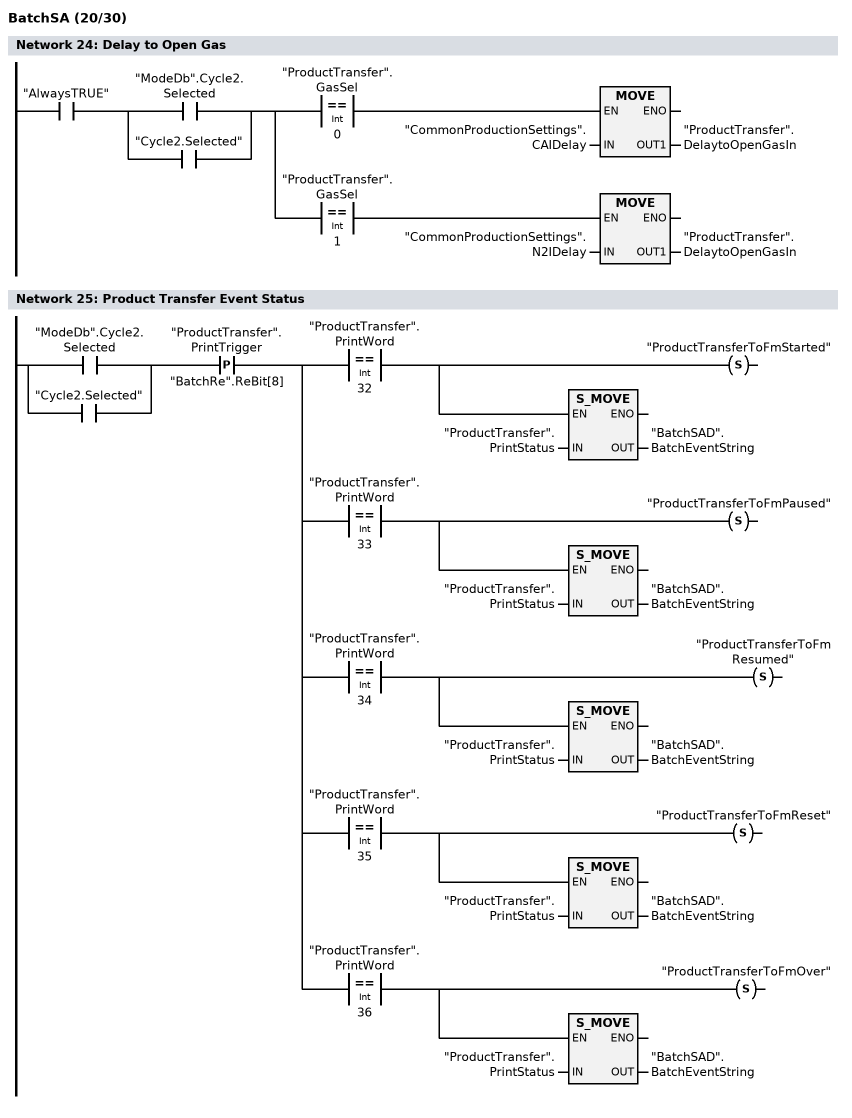
   RUNG wire#powerrail
      Contact( "AlwaysTRUE" )
      wire#w1
      Contact( "ModeDb".Cycle2.Selected )
      wire#w2
      { S7_Templates := "SrcType := Int" } EQ_Contact(in1 := "ProductTransfer".GasSel, in2 := 0)
      Move(in := "CommonProductionSettings".CAIDelay, out1 => "ProductTransfer".DelaytoOpenGasIn)
   END_RUNG
   RUNG wire#w1
      Contact( "Cycle2.Selected" )
   END_RUNG wire#w2
   RUNG wire#w2
      { S7_Templates := "SrcType := Int" } EQ_Contact(in1 := "ProductTransfer".GasSel, in2 := 1)
      Move(in := "CommonProductionSettings".N2IDelay, out1 => "ProductTransfer".DelaytoOpenGasIn)
   END_RUNG
   // the same network as SCL:
   #_w1 := "AlwaysTRUE" AND ("ModeDb".Cycle2.Selected OR "Cycle2.Selected");
   IF #_w1 AND ("ProductTransfer".GasSel = 0) THEN
       "ProductTransfer".DelaytoOpenGasIn := "CommonProductionSettings".CAIDelay;
   END_IF;
   IF #_w1 AND ("ProductTransfer".GasSel = 1) THEN
       "ProductTransfer".DelaytoOpenGasIn := "CommonProductionSettings".N2IDelay;
   END_IF;
END_REGION

REGION Network 25: Product Transfer Event Status
   RUNG wire#powerrail
      Contact( "ModeDb".Cycle2.Selected )
      wire#w1
      P_Contact(operand := "ProductTransfer".PrintTrigger, bit := "BatchRe".ReBit[8])
      wire#w2
      { S7_Templates := "SrcType := Int" } EQ_Contact(in1 := "ProductTransfer".PrintWord, in2 := 32)
      wire#w3
      S_Coil( "ProductTransferToFmStarted" )
   END_RUNG
   RUNG wire#powerrail
      Contact( "Cycle2.Selected" )
   END_RUNG wire#w1
   RUNG wire#w3
      S_Move(in := "ProductTransfer".PrintStatus, out => "BatchSAD".BatchEventString)
   END_RUNG
   RUNG wire#w2
      { S7_Templates := "SrcType := Int" } EQ_Contact(in1 := "ProductTransfer".PrintWord, in2 := 33)
      wire#w4
      S_Coil( "ProductTransferToFmPaused" )
   END_RUNG
   RUNG wire#w4
      S_Move(in := "ProductTransfer".PrintStatus, out => "BatchSAD".BatchEventString)
   END_RUNG
   RUNG wire#w2
      { S7_Templates := "SrcType := Int" } EQ_Contact(in1 := "ProductTransfer".PrintWord, in2 := 34)
      wire#w5
      S_Coil( "ProductTransferToFmResumed" )
   END_RUNG
   RUNG wire#w5
      S_Move(in := "ProductTransfer".PrintStatus, out => "BatchSAD".BatchEventString)
   END_RUNG
   RUNG wire#w2
      { S7_Templates := "SrcType := Int" } EQ_Contact(in1 := "ProductTransfer".PrintWord, in2 := 35)
      wire#w6
      S_Coil( "ProductTransferToFmReset" )
   END_RUNG
   RUNG wire#w6
      S_Move(in := "ProductTransfer".PrintStatus, out => "BatchSAD".BatchEventString)
   END_RUNG
   RUNG wire#w2
      { S7_Templates := "SrcType := Int" } EQ_Contact(in1 := "ProductTransfer".PrintWord, in2 := 36)
      wire#w7
      S_Coil( "ProductTransferToFmOver" )
   END_RUNG
   RUNG wire#w7
      S_Move(in := "ProductTransfer".PrintStatus, out => "BatchSAD".BatchEventString)
   END_RUNG
   // the same network as SCL:
   #_w1 := ("ModeDb".Cycle2.Selected OR "Cycle2.Selected") AND "ProductTransfer".PrintTrigger AND NOT "BatchRe".ReBit[8];   // rising edge of "ProductTransfer".PrintTrigger
   "BatchRe".ReBit[8] := "ProductTransfer".PrintTrigger;
   IF #_w1 AND ("ProductTransfer".PrintWord = 32) THEN
       "ProductTransferToFmStarted" := TRUE;
       "BatchSAD".BatchEventString := "ProductTransfer".PrintStatus;
   END_IF;
   IF #_w1 AND ("ProductTransfer".PrintWord = 33) THEN
       "ProductTransferToFmPaused" := TRUE;
       "BatchSAD".BatchEventString := "ProductTransfer".PrintStatus;
   END_IF;
   IF #_w1 AND ("ProductTransfer".PrintWord = 34) THEN
       "ProductTransferToFmResumed" := TRUE;
       "BatchSAD".BatchEventString := "ProductTransfer".PrintStatus;
   END_IF;
   IF #_w1 AND ("ProductTransfer".PrintWord = 35) THEN
       "ProductTransferToFmReset" := TRUE;
       "BatchSAD".BatchEventString := "ProductTransfer".PrintStatus;
   END_IF;
   IF #_w1 AND ("ProductTransfer".PrintWord = 36) THEN
       "ProductTransferToFmOver" := TRUE;
       "BatchSAD".BatchEventString := "ProductTransfer".PrintStatus;
   END_IF;
END_REGION

REGION Network 26: ******************************Jacket Vent******************************
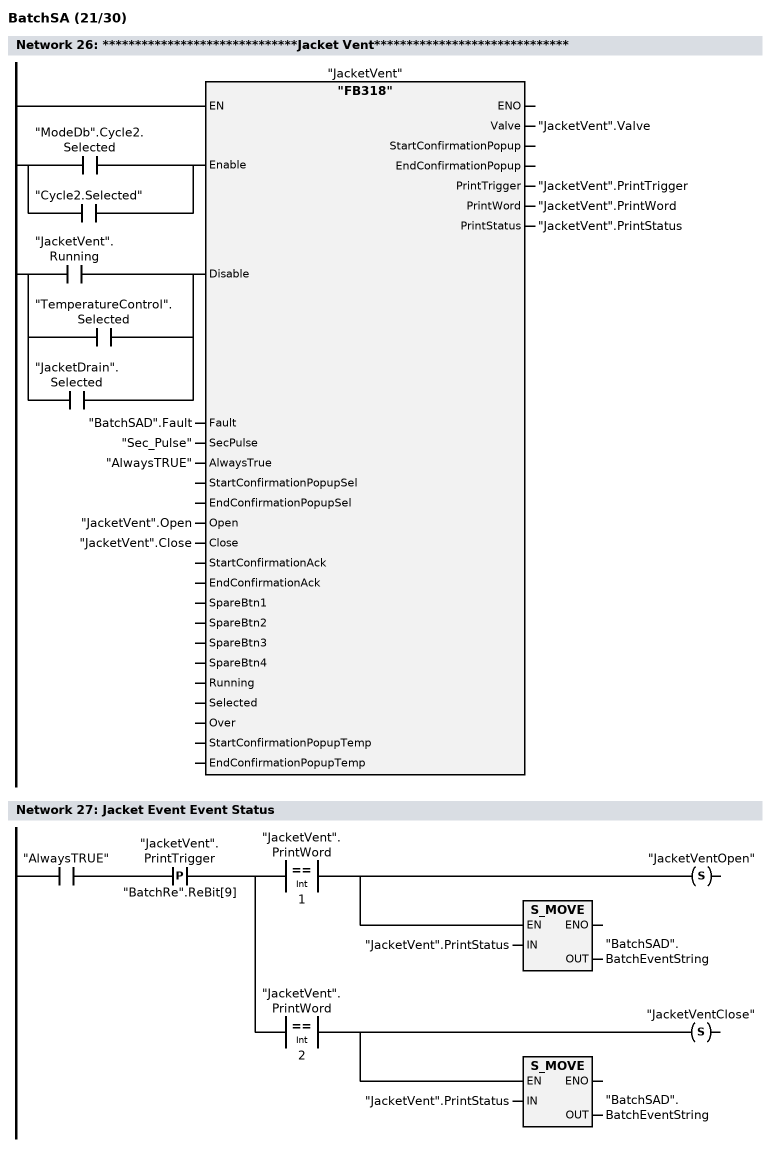
   RUNG wire#powerrail
      "JacketVent"(Enable := wire#w1, Disable := wire#w2, Fault := "BatchSAD".Fault, SecPulse := "Sec_Pulse", AlwaysTrue := "AlwaysTRUE", StartConfirmationPopupSel :=, EndConfirmationPopupSel :=, Open := "JacketVent".Open, Close := "JacketVent".Close, StartConfirmationAck :=, EndConfirmationAck :=, SpareBtn1 :=, SpareBtn2 :=, SpareBtn3 :=, SpareBtn4 :=, Running :=, Selected :=, Over :=, StartConfirmationPopupTemp :=, EndConfirmationPopupTemp :=, Valve => "JacketVent".Valve, StartConfirmationPopup =>, EndConfirmationPopup =>, PrintTrigger => "JacketVent".PrintTrigger, PrintWord => "JacketVent".PrintWord, PrintStatus => "JacketVent".PrintStatus)
   END_RUNG
   RUNG wire#powerrail
      Contact( "ModeDb".Cycle2.Selected )
   END_RUNG wire#w1
   RUNG wire#powerrail
      Contact( "Cycle2.Selected" )
   END_RUNG wire#w1
   RUNG wire#powerrail
      Contact( "JacketVent".Running )
   END_RUNG wire#w2
   RUNG wire#powerrail
      Contact( "TemperatureControl".Selected )
   END_RUNG wire#w2
   RUNG wire#powerrail
      Contact( "JacketDrain".Selected )
   END_RUNG wire#w2
   // the same network as SCL:
   "JacketVent"(Enable := "ModeDb".Cycle2.Selected OR "Cycle2.Selected",   // "FB318"
                Disable := "JacketVent".Running OR "TemperatureControl".Selected OR "JacketDrain".Selected,
                Fault := "BatchSAD".Fault,
                SecPulse := "Sec_Pulse",
                AlwaysTrue := "AlwaysTRUE",
                Open := "JacketVent".Open,
                Close := "JacketVent".Close,
                Valve => "JacketVent".Valve,
                PrintTrigger => "JacketVent".PrintTrigger,
                PrintWord => "JacketVent".PrintWord,
                PrintStatus => "JacketVent".PrintStatus);
END_REGION

REGION Network 27: Jacket Event Event Status
   RUNG wire#powerrail
      Contact( "AlwaysTRUE" )
      P_Contact(operand := "JacketVent".PrintTrigger, bit := "BatchRe".ReBit[9])
      wire#w1
      { S7_Templates := "SrcType := Int" } EQ_Contact(in1 := "JacketVent".PrintWord, in2 := 1)
      wire#w2
      S_Coil( "JacketVentOpen" )
   END_RUNG
   RUNG wire#w2
      S_Move(in := "JacketVent".PrintStatus, out => "BatchSAD".BatchEventString)
   END_RUNG
   RUNG wire#w1
      { S7_Templates := "SrcType := Int" } EQ_Contact(in1 := "JacketVent".PrintWord, in2 := 2)
      wire#w3
      S_Coil( "JacketVentClose" )
   END_RUNG
   RUNG wire#w3
      S_Move(in := "JacketVent".PrintStatus, out => "BatchSAD".BatchEventString)
   END_RUNG
   // the same network as SCL:
   #_w1 := "AlwaysTRUE" AND "JacketVent".PrintTrigger AND NOT "BatchRe".ReBit[9];   // rising edge of "JacketVent".PrintTrigger
   "BatchRe".ReBit[9] := "JacketVent".PrintTrigger;
   IF #_w1 AND ("JacketVent".PrintWord = 1) THEN
       "JacketVentOpen" := TRUE;
       "BatchSAD".BatchEventString := "JacketVent".PrintStatus;
   END_IF;
   IF #_w1 AND ("JacketVent".PrintWord = 2) THEN
       "JacketVentClose" := TRUE;
       "BatchSAD".BatchEventString := "JacketVent".PrintStatus;
   END_IF;
END_REGION

REGION Network 28: ******************************Jacket Drain******************************
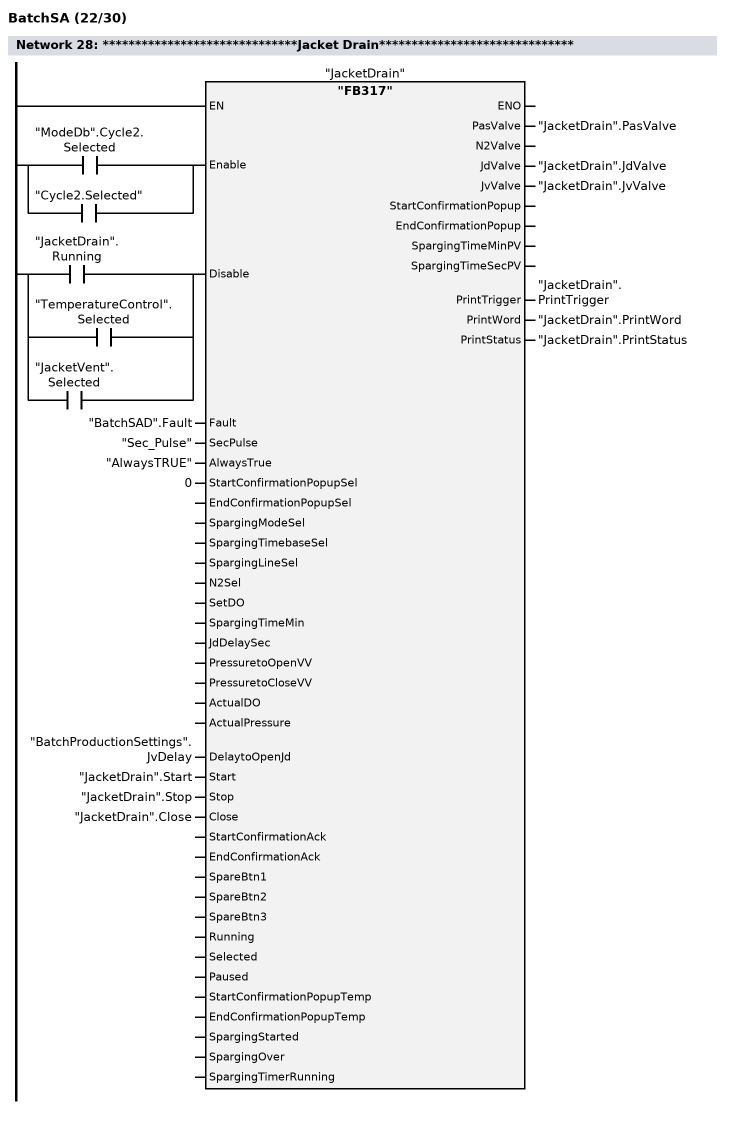
   RUNG wire#powerrail
      "JacketDrain"(Enable := wire#w1, Disable := wire#w2, Fault := "BatchSAD".Fault, SecPulse := "Sec_Pulse", AlwaysTrue := "AlwaysTRUE", StartConfirmationPopupSel := 0, EndConfirmationPopupSel :=, SpargingModeSel :=, SpargingTimebaseSel :=, SpargingLineSel :=, N2Sel :=, SetDO :=, SpargingTimeMin :=, JdDelaySec :=, PressuretoOpenVV :=, PressuretoCloseVV :=, ActualDO :=, ActualPressure :=, DelaytoOpenJd := "BatchProductionSettings".JvDelay, Start := "JacketDrain".Start, Stop := "JacketDrain".Stop, Close := "JacketDrain".Close, StartConfirmationAck :=, EndConfirmationAck :=, SpareBtn1 :=, SpareBtn2 :=, SpareBtn3 :=, Running :=, Selected :=, Paused :=, StartConfirmationPopupTemp :=, EndConfirmationPopupTemp :=, SpargingStarted :=, SpargingOver :=, SpargingTimerRunning :=, PasValve => "JacketDrain".PasValve, N2Valve =>, JdValve => "JacketDrain".JdValve, JvValve => "JacketDrain".JvValve, StartConfirmationPopup =>, EndConfirmationPopup =>, SpargingTimeMinPV =>, SpargingTimeSecPV =>, PrintTrigger => "JacketDrain".PrintTrigger, PrintWord => "JacketDrain".PrintWord, PrintStatus => "JacketDrain".PrintStatus)
   END_RUNG
   RUNG wire#powerrail
      Contact( "ModeDb".Cycle2.Selected )
   END_RUNG wire#w1
   RUNG wire#powerrail
      Contact( "Cycle2.Selected" )
   END_RUNG wire#w1
   RUNG wire#powerrail
      Contact( "JacketDrain".Running )
   END_RUNG wire#w2
   RUNG wire#powerrail
      Contact( "TemperatureControl".Selected )
   END_RUNG wire#w2
   RUNG wire#powerrail
      Contact( "JacketVent".Selected )
   END_RUNG wire#w2
   // the same network as SCL:
   "JacketDrain"(Enable := "ModeDb".Cycle2.Selected OR "Cycle2.Selected",   // "FB317"
                 Disable := "JacketDrain".Running OR "TemperatureControl".Selected OR "JacketVent".Selected,
                 Fault := "BatchSAD".Fault,
                 SecPulse := "Sec_Pulse",
                 AlwaysTrue := "AlwaysTRUE",
                 StartConfirmationPopupSel := 0,
                 DelaytoOpenJd := "BatchProductionSettings".JvDelay,
                 Start := "JacketDrain".Start,
                 Stop := "JacketDrain".Stop,
                 Close := "JacketDrain".Close,
                 PasValve => "JacketDrain".PasValve,
                 JdValve => "JacketDrain".JdValve,
                 JvValve => "JacketDrain".JvValve,
                 PrintTrigger => "JacketDrain".PrintTrigger,
                 PrintWord => "JacketDrain".PrintWord,
                 PrintStatus => "JacketDrain".PrintStatus);
END_REGION

REGION Network 29: Jacket Drain Event Status
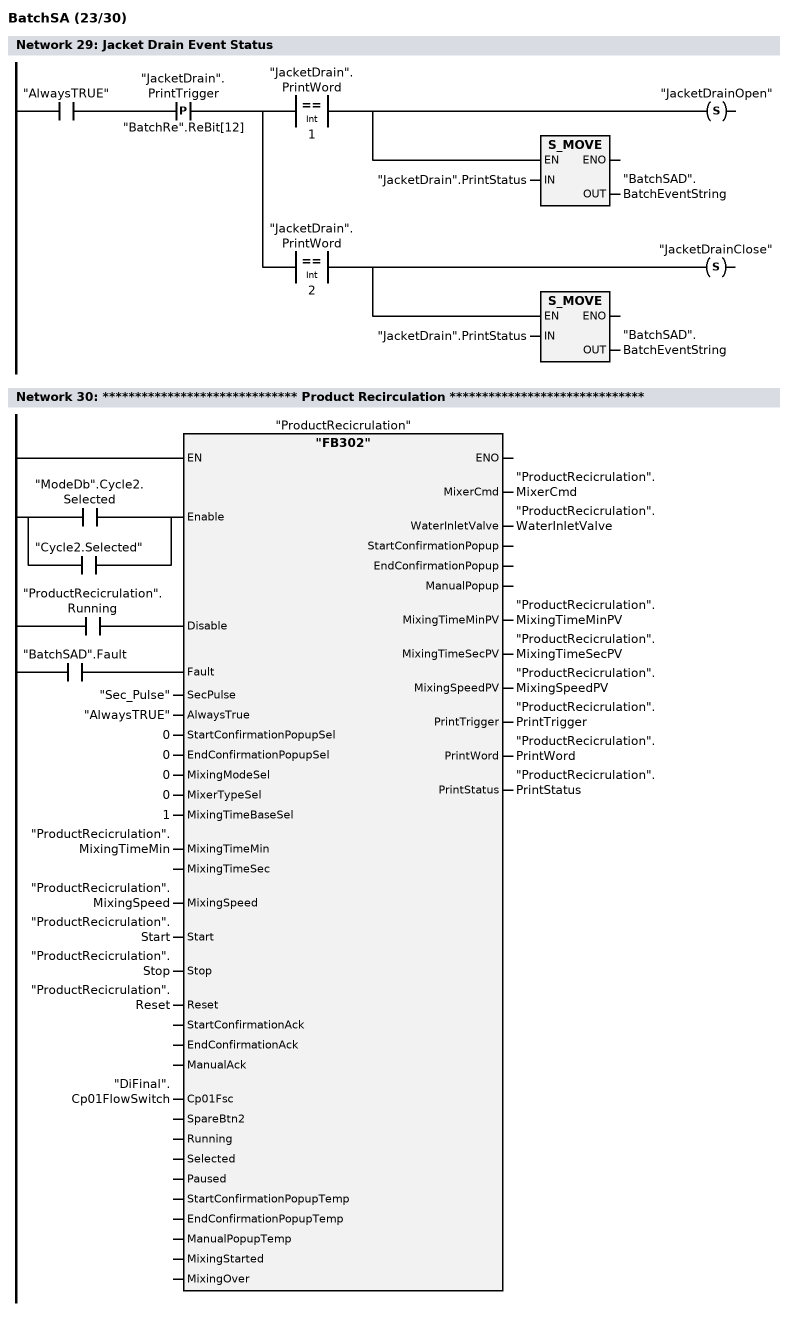
   RUNG wire#powerrail
      Contact( "AlwaysTRUE" )
      P_Contact(operand := "JacketDrain".PrintTrigger, bit := "BatchRe".ReBit[12])
      wire#w1
      { S7_Templates := "SrcType := Int" } EQ_Contact(in1 := "JacketDrain".PrintWord, in2 := 1)
      wire#w2
      S_Coil( "JacketDrainOpen" )
   END_RUNG
   RUNG wire#w2
      S_Move(in := "JacketDrain".PrintStatus, out => "BatchSAD".BatchEventString)
   END_RUNG
   RUNG wire#w1
      { S7_Templates := "SrcType := Int" } EQ_Contact(in1 := "JacketDrain".PrintWord, in2 := 2)
      wire#w3
      S_Coil( "JacketDrainClose" )
   END_RUNG
   RUNG wire#w3
      S_Move(in := "JacketDrain".PrintStatus, out => "BatchSAD".BatchEventString)
   END_RUNG
   // the same network as SCL:
   #_w1 := "AlwaysTRUE" AND "JacketDrain".PrintTrigger AND NOT "BatchRe".ReBit[12];   // rising edge of "JacketDrain".PrintTrigger
   "BatchRe".ReBit[12] := "JacketDrain".PrintTrigger;
   IF #_w1 AND ("JacketDrain".PrintWord = 1) THEN
       "JacketDrainOpen" := TRUE;
       "BatchSAD".BatchEventString := "JacketDrain".PrintStatus;
   END_IF;
   IF #_w1 AND ("JacketDrain".PrintWord = 2) THEN
       "JacketDrainClose" := TRUE;
       "BatchSAD".BatchEventString := "JacketDrain".PrintStatus;
   END_IF;
END_REGION

REGION Network 30: ****************************** Product Recirculation ******************************
   RUNG wire#powerrail
      "ProductRecicrulation"(Enable := wire#w1, Disable := wire#w2, Fault := wire#w3, SecPulse := "Sec_Pulse", AlwaysTrue := "AlwaysTRUE", StartConfirmationPopupSel := 0, EndConfirmationPopupSel := 0, MixingModeSel := 0, MixerTypeSel := 0, MixingTimeBaseSel := 1, MixingTimeMin := "ProductRecicrulation".MixingTimeMin, MixingTimeSec :=, MixingSpeed := "ProductRecicrulation".MixingSpeed, Start := "ProductRecicrulation".Start, Stop := "ProductRecicrulation".Stop, Reset := "ProductRecicrulation".Reset, StartConfirmationAck :=, EndConfirmationAck :=, ManualAck :=, Cp01Fsc := "DiFinal".Cp01FlowSwitch, SpareBtn2 :=, Running :=, Selected :=, Paused :=, StartConfirmationPopupTemp :=, EndConfirmationPopupTemp :=, ManualPopupTemp :=, MixingStarted :=, MixingOver :=, MixerCmd => "ProductRecicrulation".MixerCmd, WaterInletValve => "ProductRecicrulation".WaterInletValve, StartConfirmationPopup =>, EndConfirmationPopup =>, ManualPopup =>, MixingTimeMinPV => "ProductRecicrulation".MixingTimeMinPV, MixingTimeSecPV => "ProductRecicrulation".MixingTimeSecPV, MixingSpeedPV => "ProductRecicrulation".MixingSpeedPV, PrintTrigger => "ProductRecicrulation".PrintTrigger, PrintWord => "ProductRecicrulation".PrintWord, PrintStatus => "ProductRecicrulation".PrintStatus)
   END_RUNG
   RUNG wire#powerrail
      Contact( "ModeDb".Cycle2.Selected )
   END_RUNG wire#w1
   RUNG wire#powerrail
      Contact( "Cycle2.Selected" )
   END_RUNG wire#w1
   RUNG wire#powerrail
      Contact( "ProductRecicrulation".Running )
   END_RUNG wire#w2
   RUNG wire#powerrail
      Contact( "BatchSAD".Fault )
   END_RUNG wire#w3
   // the same network as SCL:
   "ProductRecicrulation"(Enable := "ModeDb".Cycle2.Selected OR "Cycle2.Selected",   // "FB302"
                          Disable := "ProductRecicrulation".Running,
                          Fault := "BatchSAD".Fault,
                          SecPulse := "Sec_Pulse",
                          AlwaysTrue := "AlwaysTRUE",
                          StartConfirmationPopupSel := 0,
                          EndConfirmationPopupSel := 0,
                          MixingModeSel := 0,
                          MixerTypeSel := 0,
                          MixingTimeBaseSel := 1,
                          MixingTimeMin := "ProductRecicrulation".MixingTimeMin,
                          MixingSpeed := "ProductRecicrulation".MixingSpeed,
                          Start := "ProductRecicrulation".Start,
                          Stop := "ProductRecicrulation".Stop,
                          Reset := "ProductRecicrulation".Reset,
                          Cp01Fsc := "DiFinal".Cp01FlowSwitch,
                          MixerCmd => "ProductRecicrulation".MixerCmd,
                          WaterInletValve => "ProductRecicrulation".WaterInletValve,
                          MixingTimeMinPV => "ProductRecicrulation".MixingTimeMinPV,
                          MixingTimeSecPV => "ProductRecicrulation".MixingTimeSecPV,
                          MixingSpeedPV => "ProductRecicrulation".MixingSpeedPV,
                          PrintTrigger => "ProductRecicrulation".PrintTrigger,
                          PrintWord => "ProductRecicrulation".PrintWord,
                          PrintStatus => "ProductRecicrulation".PrintStatus);
END_REGION

REGION Network 31: Mm01 Mixing Event Staus
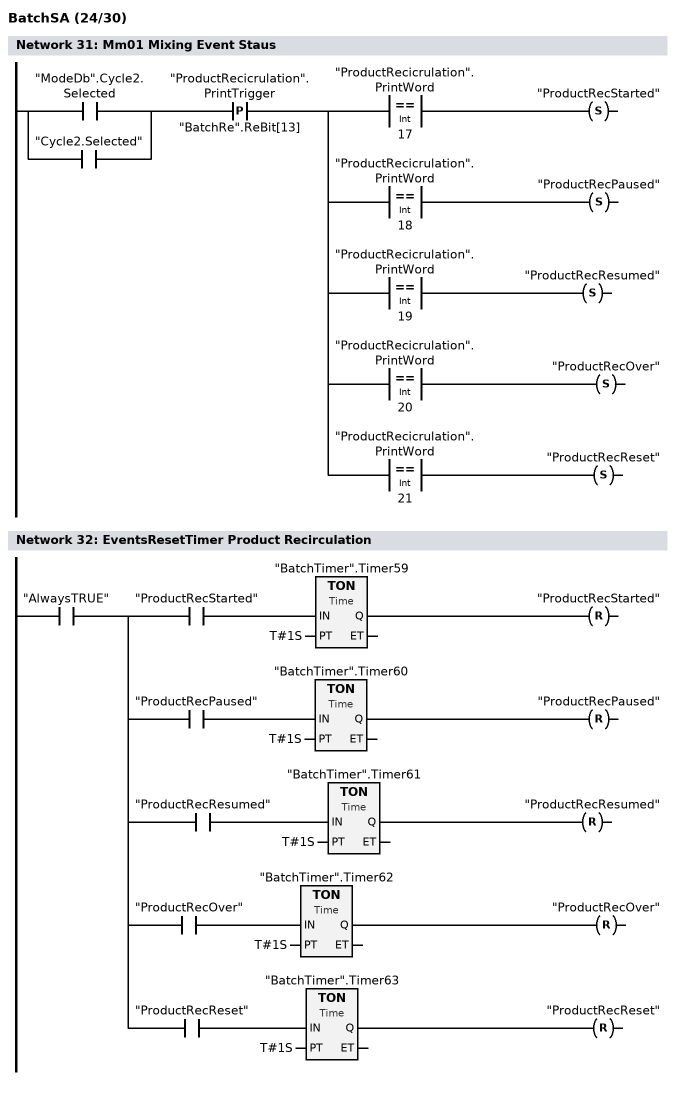
   RUNG wire#powerrail
      Contact( "ModeDb".Cycle2.Selected )
      wire#w1
      P_Contact(operand := "ProductRecicrulation".PrintTrigger, bit := "BatchRe".ReBit[13])
      wire#w2
      { S7_Templates := "SrcType := Int" } EQ_Contact(in1 := "ProductRecicrulation".PrintWord, in2 := 17)
      S_Coil( "ProductRecStarted" )
   END_RUNG
   RUNG wire#powerrail
      Contact( "Cycle2.Selected" )
   END_RUNG wire#w1
   RUNG wire#w2
      { S7_Templates := "SrcType := Int" } EQ_Contact(in1 := "ProductRecicrulation".PrintWord, in2 := 18)
      S_Coil( "ProductRecPaused" )
   END_RUNG
   RUNG wire#w2
      { S7_Templates := "SrcType := Int" } EQ_Contact(in1 := "ProductRecicrulation".PrintWord, in2 := 19)
      S_Coil( "ProductRecResumed" )
   END_RUNG
   RUNG wire#w2
      { S7_Templates := "SrcType := Int" } EQ_Contact(in1 := "ProductRecicrulation".PrintWord, in2 := 20)
      S_Coil( "ProductRecOver" )
   END_RUNG
   RUNG wire#w2
      { S7_Templates := "SrcType := Int" } EQ_Contact(in1 := "ProductRecicrulation".PrintWord, in2 := 21)
      S_Coil( "ProductRecReset" )
   END_RUNG
   // the same network as SCL:
   #_w1 := ("ModeDb".Cycle2.Selected OR "Cycle2.Selected") AND "ProductRecicrulation".PrintTrigger AND NOT "BatchRe".ReBit[13];   // rising edge of "ProductRecicrulation".PrintTrigger
   "BatchRe".ReBit[13] := "ProductRecicrulation".PrintTrigger;
   IF #_w1 AND ("ProductRecicrulation".PrintWord = 17) THEN "ProductRecStarted" := TRUE; END_IF;
   IF #_w1 AND ("ProductRecicrulation".PrintWord = 18) THEN "ProductRecPaused" := TRUE; END_IF;
   IF #_w1 AND ("ProductRecicrulation".PrintWord = 19) THEN "ProductRecResumed" := TRUE; END_IF;
   IF #_w1 AND ("ProductRecicrulation".PrintWord = 20) THEN "ProductRecOver" := TRUE; END_IF;
   IF #_w1 AND ("ProductRecicrulation".PrintWord = 21) THEN "ProductRecReset" := TRUE; END_IF;
END_REGION

REGION Network 32: EventsResetTimer Product Recirculation
   RUNG wire#powerrail
      Contact( "AlwaysTRUE" )
      wire#w1
      Contact( "ProductRecStarted" )
      { S7_Templates := "time_type := Time" } "BatchTimer".Timer59.TON(pt := T#1S, et =>)
      R_Coil( "ProductRecStarted" )
   END_RUNG
   RUNG wire#w1
      Contact( "ProductRecPaused" )
      { S7_Templates := "time_type := Time" } "BatchTimer".Timer60.TON(pt := T#1S, et =>)
      R_Coil( "ProductRecPaused" )
   END_RUNG
   RUNG wire#w1
      Contact( "ProductRecResumed" )
      { S7_Templates := "time_type := Time" } "BatchTimer".Timer61.TON(pt := T#1S, et =>)
      R_Coil( "ProductRecResumed" )
   END_RUNG
   RUNG wire#w1
      Contact( "ProductRecOver" )
      { S7_Templates := "time_type := Time" } "BatchTimer".Timer62.TON(pt := T#1S, et =>)
      R_Coil( "ProductRecOver" )
   END_RUNG
   RUNG wire#w1
      Contact( "ProductRecReset" )
      { S7_Templates := "time_type := Time" } "BatchTimer".Timer63.TON(pt := T#1S, et =>)
      R_Coil( "ProductRecReset" )
   END_RUNG
   // the same network as SCL:
   "BatchTimer".Timer59.TON(IN := "AlwaysTRUE" AND "ProductRecStarted", PT := T#1S);
   IF "BatchTimer".Timer59.Q THEN "ProductRecStarted" := FALSE; END_IF;
   "BatchTimer".Timer60.TON(IN := "AlwaysTRUE" AND "ProductRecPaused", PT := T#1S);
   IF "BatchTimer".Timer60.Q THEN "ProductRecPaused" := FALSE; END_IF;
   "BatchTimer".Timer61.TON(IN := "AlwaysTRUE" AND "ProductRecResumed", PT := T#1S);
   IF "BatchTimer".Timer61.Q THEN "ProductRecResumed" := FALSE; END_IF;
   "BatchTimer".Timer62.TON(IN := "AlwaysTRUE" AND "ProductRecOver", PT := T#1S);
   IF "BatchTimer".Timer62.Q THEN "ProductRecOver" := FALSE; END_IF;
   "BatchTimer".Timer63.TON(IN := "AlwaysTRUE" AND "ProductRecReset", PT := T#1S);
   IF "BatchTimer".Timer63.Q THEN "ProductRecReset" := FALSE; END_IF;
END_REGION

REGION Network 33: EventsResetTimer FIill PWI
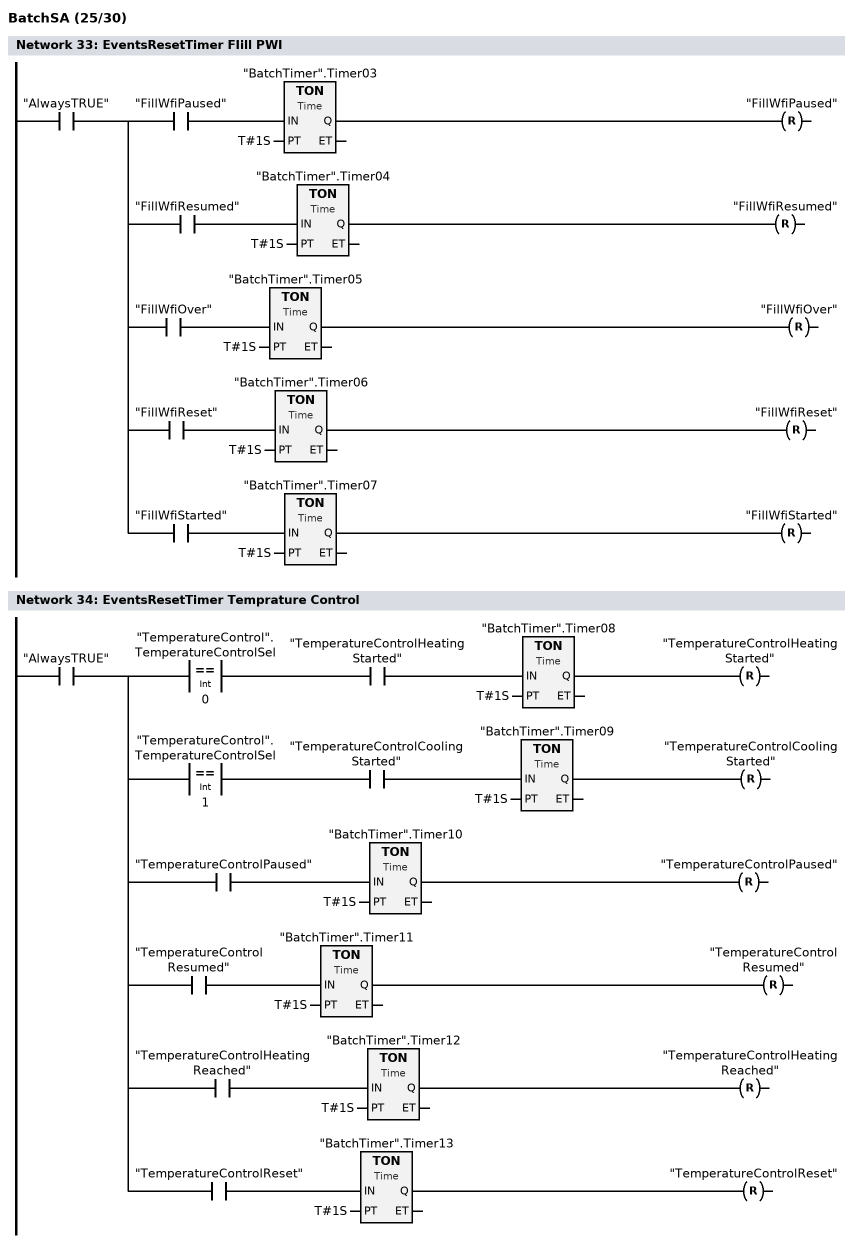
   RUNG wire#powerrail
      Contact( "AlwaysTRUE" )
      wire#w1
      Contact( "FillWfiPaused" )
      { S7_Templates := "time_type := Time" } "BatchTimer".Timer03.TON(pt := T#1S, et =>)
      R_Coil( "FillWfiPaused" )
   END_RUNG
   RUNG wire#w1
      Contact( "FillWfiResumed" )
      { S7_Templates := "time_type := Time" } "BatchTimer".Timer04.TON(pt := T#1S, et =>)
      R_Coil( "FillWfiResumed" )
   END_RUNG
   RUNG wire#w1
      Contact( "FillWfiOver" )
      { S7_Templates := "time_type := Time" } "BatchTimer".Timer05.TON(pt := T#1S, et =>)
      R_Coil( "FillWfiOver" )
   END_RUNG
   RUNG wire#w1
      Contact( "FillWfiReset" )
      { S7_Templates := "time_type := Time" } "BatchTimer".Timer06.TON(pt := T#1S, et =>)
      R_Coil( "FillWfiReset" )
   END_RUNG
   RUNG wire#w1
      Contact( "FillWfiStarted" )
      { S7_Templates := "time_type := Time" } "BatchTimer".Timer07.TON(pt := T#1S, et =>)
      R_Coil( "FillWfiStarted" )
   END_RUNG
   // the same network as SCL:
   "BatchTimer".Timer03.TON(IN := "AlwaysTRUE" AND "FillWfiPaused", PT := T#1S);
   IF "BatchTimer".Timer03.Q THEN "FillWfiPaused" := FALSE; END_IF;
   "BatchTimer".Timer04.TON(IN := "AlwaysTRUE" AND "FillWfiResumed", PT := T#1S);
   IF "BatchTimer".Timer04.Q THEN "FillWfiResumed" := FALSE; END_IF;
   "BatchTimer".Timer05.TON(IN := "AlwaysTRUE" AND "FillWfiOver", PT := T#1S);
   IF "BatchTimer".Timer05.Q THEN "FillWfiOver" := FALSE; END_IF;
   "BatchTimer".Timer06.TON(IN := "AlwaysTRUE" AND "FillWfiReset", PT := T#1S);
   IF "BatchTimer".Timer06.Q THEN "FillWfiReset" := FALSE; END_IF;
   "BatchTimer".Timer07.TON(IN := "AlwaysTRUE" AND "FillWfiStarted", PT := T#1S);
   IF "BatchTimer".Timer07.Q THEN "FillWfiStarted" := FALSE; END_IF;
END_REGION

REGION Network 34: EventsResetTimer Temprature Control
   RUNG wire#powerrail
      Contact( "AlwaysTRUE" )
      wire#w1
      { S7_Templates := "SrcType := Int" } EQ_Contact(in1 := "TemperatureControl".TemperatureControlSel, in2 := 0)
      Contact( "TemperatureControlHeatingStarted" )
      { S7_Templates := "time_type := Time" } "BatchTimer".Timer08.TON(pt := T#1S, et =>)
      R_Coil( "TemperatureControlHeatingStarted" )
   END_RUNG
   RUNG wire#w1
      { S7_Templates := "SrcType := Int" } EQ_Contact(in1 := "TemperatureControl".TemperatureControlSel, in2 := 1)
      Contact( "TemperatureControlCoolingStarted" )
      { S7_Templates := "time_type := Time" } "BatchTimer".Timer09.TON(pt := T#1S, et =>)
      R_Coil( "TemperatureControlCoolingStarted" )
   END_RUNG
   RUNG wire#w1
      Contact( "TemperatureControlPaused" )
      { S7_Templates := "time_type := Time" } "BatchTimer".Timer10.TON(pt := T#1S, et =>)
      R_Coil( "TemperatureControlPaused" )
   END_RUNG
   RUNG wire#w1
      Contact( "TemperatureControlResumed" )
      { S7_Templates := "time_type := Time" } "BatchTimer".Timer11.TON(pt := T#1S, et =>)
      R_Coil( "TemperatureControlResumed" )
   END_RUNG
   RUNG wire#w1
      Contact( "TemperatureControlHeatingReached" )
      { S7_Templates := "time_type := Time" } "BatchTimer".Timer12.TON(pt := T#1S, et =>)
      R_Coil( "TemperatureControlHeatingReached" )
   END_RUNG
   RUNG wire#w1
      Contact( "TemperatureControlReset" )
      { S7_Templates := "time_type := Time" } "BatchTimer".Timer13.TON(pt := T#1S, et =>)
      R_Coil( "TemperatureControlReset" )
   END_RUNG
   // the same network as SCL:
   "BatchTimer".Timer08.TON(IN := "AlwaysTRUE" AND ("TemperatureControl".TemperatureControlSel = 0) AND "TemperatureControlHeatingStarted",
                           PT := T#1S);
   IF "BatchTimer".Timer08.Q THEN "TemperatureControlHeatingStarted" := FALSE; END_IF;
   "BatchTimer".Timer09.TON(IN := "AlwaysTRUE" AND ("TemperatureControl".TemperatureControlSel = 1) AND "TemperatureControlCoolingStarted",
                           PT := T#1S);
   IF "BatchTimer".Timer09.Q THEN "TemperatureControlCoolingStarted" := FALSE; END_IF;
   "BatchTimer".Timer10.TON(IN := "AlwaysTRUE" AND "TemperatureControlPaused", PT := T#1S);
   IF "BatchTimer".Timer10.Q THEN "TemperatureControlPaused" := FALSE; END_IF;
   "BatchTimer".Timer11.TON(IN := "AlwaysTRUE" AND "TemperatureControlResumed", PT := T#1S);
   IF "BatchTimer".Timer11.Q THEN "TemperatureControlResumed" := FALSE; END_IF;
   "BatchTimer".Timer12.TON(IN := "AlwaysTRUE" AND "TemperatureControlHeatingReached", PT := T#1S);
   IF "BatchTimer".Timer12.Q THEN "TemperatureControlHeatingReached" := FALSE; END_IF;
   "BatchTimer".Timer13.TON(IN := "AlwaysTRUE" AND "TemperatureControlReset", PT := T#1S);
   IF "BatchTimer".Timer13.Q THEN "TemperatureControlReset" := FALSE; END_IF;
END_REGION

REGION Network 35: EventsResetTimer RawMaterialAddition
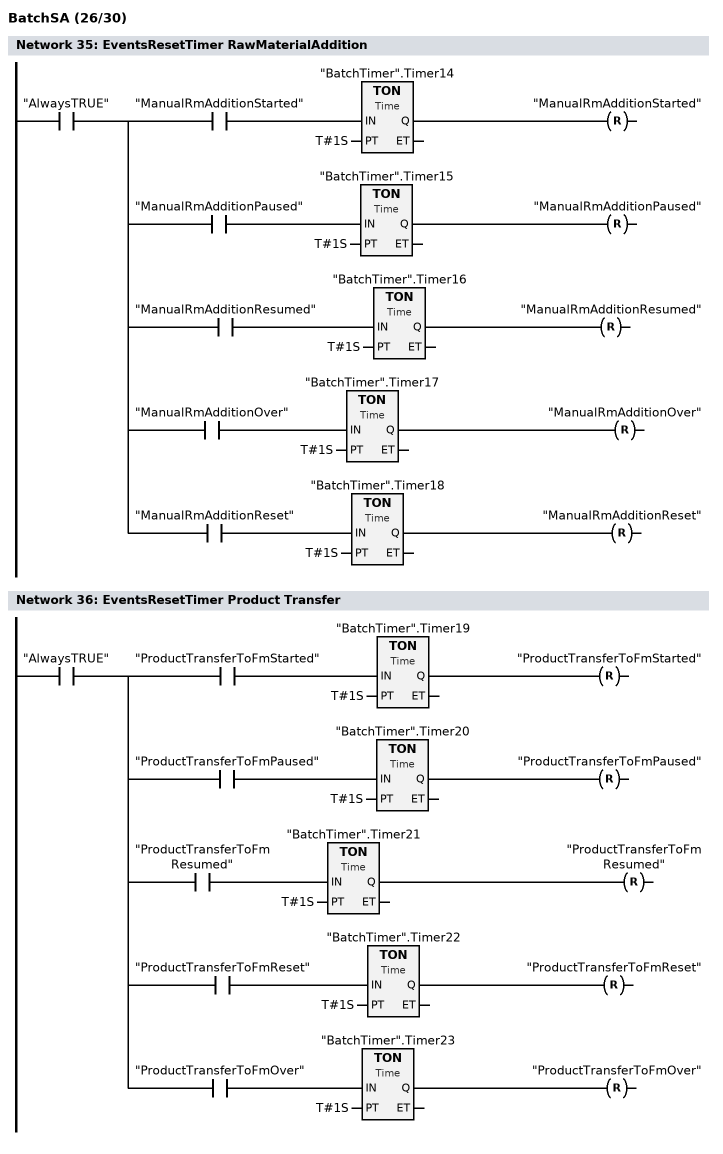
   RUNG wire#powerrail
      Contact( "AlwaysTRUE" )
      wire#w1
      Contact( "ManualRmAdditionStarted" )
      { S7_Templates := "time_type := Time" } "BatchTimer".Timer14.TON(pt := T#1S, et =>)
      R_Coil( "ManualRmAdditionStarted" )
   END_RUNG
   RUNG wire#w1
      Contact( "ManualRmAdditionPaused" )
      { S7_Templates := "time_type := Time" } "BatchTimer".Timer15.TON(pt := T#1S, et =>)
      R_Coil( "ManualRmAdditionPaused" )
   END_RUNG
   RUNG wire#w1
      Contact( "ManualRmAdditionResumed" )
      { S7_Templates := "time_type := Time" } "BatchTimer".Timer16.TON(pt := T#1S, et =>)
      R_Coil( "ManualRmAdditionResumed" )
   END_RUNG
   RUNG wire#w1
      Contact( "ManualRmAdditionOver" )
      { S7_Templates := "time_type := Time" } "BatchTimer".Timer17.TON(pt := T#1S, et =>)
      R_Coil( "ManualRmAdditionOver" )
   END_RUNG
   RUNG wire#w1
      Contact( "ManualRmAdditionReset" )
      { S7_Templates := "time_type := Time" } "BatchTimer".Timer18.TON(pt := T#1S, et =>)
      R_Coil( "ManualRmAdditionReset" )
   END_RUNG
   // the same network as SCL:
   "BatchTimer".Timer14.TON(IN := "AlwaysTRUE" AND "ManualRmAdditionStarted", PT := T#1S);
   IF "BatchTimer".Timer14.Q THEN "ManualRmAdditionStarted" := FALSE; END_IF;
   "BatchTimer".Timer15.TON(IN := "AlwaysTRUE" AND "ManualRmAdditionPaused", PT := T#1S);
   IF "BatchTimer".Timer15.Q THEN "ManualRmAdditionPaused" := FALSE; END_IF;
   "BatchTimer".Timer16.TON(IN := "AlwaysTRUE" AND "ManualRmAdditionResumed", PT := T#1S);
   IF "BatchTimer".Timer16.Q THEN "ManualRmAdditionResumed" := FALSE; END_IF;
   "BatchTimer".Timer17.TON(IN := "AlwaysTRUE" AND "ManualRmAdditionOver", PT := T#1S);
   IF "BatchTimer".Timer17.Q THEN "ManualRmAdditionOver" := FALSE; END_IF;
   "BatchTimer".Timer18.TON(IN := "AlwaysTRUE" AND "ManualRmAdditionReset", PT := T#1S);
   IF "BatchTimer".Timer18.Q THEN "ManualRmAdditionReset" := FALSE; END_IF;
END_REGION

REGION Network 36: EventsResetTimer Product Transfer
   RUNG wire#powerrail
      Contact( "AlwaysTRUE" )
      wire#w1
      Contact( "ProductTransferToFmStarted" )
      { S7_Templates := "time_type := Time" } "BatchTimer".Timer19.TON(pt := T#1S, et =>)
      R_Coil( "ProductTransferToFmStarted" )
   END_RUNG
   RUNG wire#w1
      Contact( "ProductTransferToFmPaused" )
      { S7_Templates := "time_type := Time" } "BatchTimer".Timer20.TON(pt := T#1S, et =>)
      R_Coil( "ProductTransferToFmPaused" )
   END_RUNG
   RUNG wire#w1
      Contact( "ProductTransferToFmResumed" )
      { S7_Templates := "time_type := Time" } "BatchTimer".Timer21.TON(pt := T#1S, et =>)
      R_Coil( "ProductTransferToFmResumed" )
   END_RUNG
   RUNG wire#w1
      Contact( "ProductTransferToFmReset" )
      { S7_Templates := "time_type := Time" } "BatchTimer".Timer22.TON(pt := T#1S, et =>)
      R_Coil( "ProductTransferToFmReset" )
   END_RUNG
   RUNG wire#w1
      Contact( "ProductTransferToFmOver" )
      { S7_Templates := "time_type := Time" } "BatchTimer".Timer23.TON(pt := T#1S, et =>)
      R_Coil( "ProductTransferToFmOver" )
   END_RUNG
   // the same network as SCL:
   "BatchTimer".Timer19.TON(IN := "AlwaysTRUE" AND "ProductTransferToFmStarted", PT := T#1S);
   IF "BatchTimer".Timer19.Q THEN "ProductTransferToFmStarted" := FALSE; END_IF;
   "BatchTimer".Timer20.TON(IN := "AlwaysTRUE" AND "ProductTransferToFmPaused", PT := T#1S);
   IF "BatchTimer".Timer20.Q THEN "ProductTransferToFmPaused" := FALSE; END_IF;
   "BatchTimer".Timer21.TON(IN := "AlwaysTRUE" AND "ProductTransferToFmResumed", PT := T#1S);
   IF "BatchTimer".Timer21.Q THEN "ProductTransferToFmResumed" := FALSE; END_IF;
   "BatchTimer".Timer22.TON(IN := "AlwaysTRUE" AND "ProductTransferToFmReset", PT := T#1S);
   IF "BatchTimer".Timer22.Q THEN "ProductTransferToFmReset" := FALSE; END_IF;
   "BatchTimer".Timer23.TON(IN := "AlwaysTRUE" AND "ProductTransferToFmOver", PT := T#1S);
   IF "BatchTimer".Timer23.Q THEN "ProductTransferToFmOver" := FALSE; END_IF;
END_REGION

REGION Network 37: EventsResetTimer Mm01 Mixing
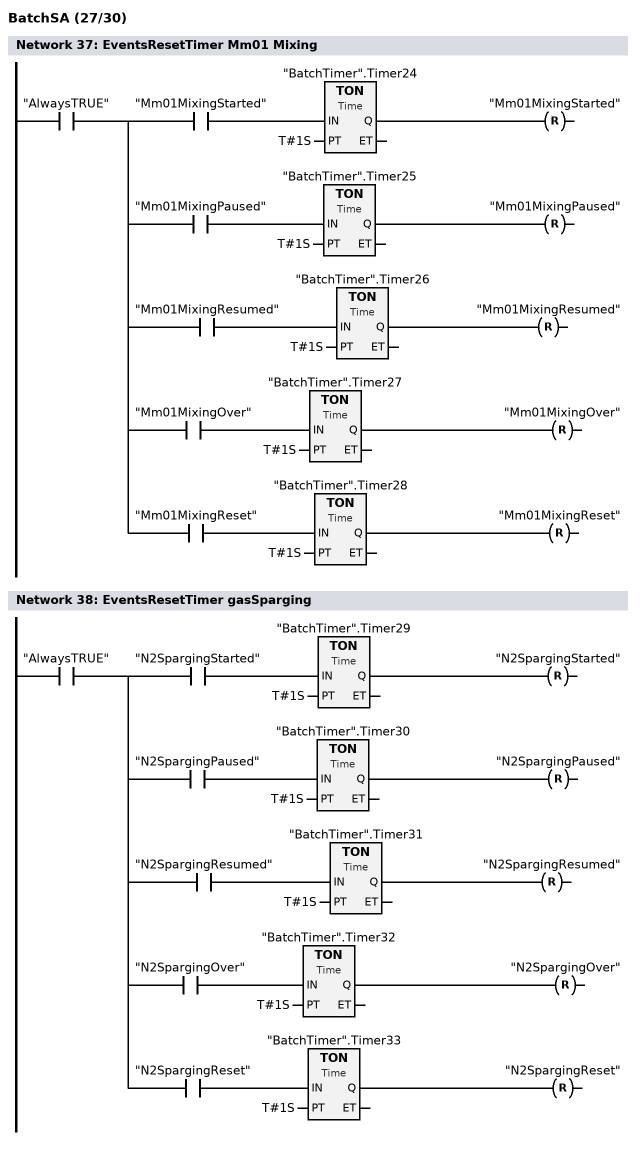
   RUNG wire#powerrail
      Contact( "AlwaysTRUE" )
      wire#w1
      Contact( "Mm01MixingStarted" )
      { S7_Templates := "time_type := Time" } "BatchTimer".Timer24.TON(pt := T#1S, et =>)
      R_Coil( "Mm01MixingStarted" )
   END_RUNG
   RUNG wire#w1
      Contact( "Mm01MixingPaused" )
      { S7_Templates := "time_type := Time" } "BatchTimer".Timer25.TON(pt := T#1S, et =>)
      R_Coil( "Mm01MixingPaused" )
   END_RUNG
   RUNG wire#w1
      Contact( "Mm01MixingResumed" )
      { S7_Templates := "time_type := Time" } "BatchTimer".Timer26.TON(pt := T#1S, et =>)
      R_Coil( "Mm01MixingResumed" )
   END_RUNG
   RUNG wire#w1
      Contact( "Mm01MixingOver" )
      { S7_Templates := "time_type := Time" } "BatchTimer".Timer27.TON(pt := T#1S, et =>)
      R_Coil( "Mm01MixingOver" )
   END_RUNG
   RUNG wire#w1
      Contact( "Mm01MixingReset" )
      { S7_Templates := "time_type := Time" } "BatchTimer".Timer28.TON(pt := T#1S, et =>)
      R_Coil( "Mm01MixingReset" )
   END_RUNG
   // the same network as SCL:
   "BatchTimer".Timer24.TON(IN := "AlwaysTRUE" AND "Mm01MixingStarted", PT := T#1S);
   IF "BatchTimer".Timer24.Q THEN "Mm01MixingStarted" := FALSE; END_IF;
   "BatchTimer".Timer25.TON(IN := "AlwaysTRUE" AND "Mm01MixingPaused", PT := T#1S);
   IF "BatchTimer".Timer25.Q THEN "Mm01MixingPaused" := FALSE; END_IF;
   "BatchTimer".Timer26.TON(IN := "AlwaysTRUE" AND "Mm01MixingResumed", PT := T#1S);
   IF "BatchTimer".Timer26.Q THEN "Mm01MixingResumed" := FALSE; END_IF;
   "BatchTimer".Timer27.TON(IN := "AlwaysTRUE" AND "Mm01MixingOver", PT := T#1S);
   IF "BatchTimer".Timer27.Q THEN "Mm01MixingOver" := FALSE; END_IF;
   "BatchTimer".Timer28.TON(IN := "AlwaysTRUE" AND "Mm01MixingReset", PT := T#1S);
   IF "BatchTimer".Timer28.Q THEN "Mm01MixingReset" := FALSE; END_IF;
END_REGION

REGION Network 38: EventsResetTimer gasSparging
   RUNG wire#powerrail
      Contact( "AlwaysTRUE" )
      wire#w1
      Contact( "N2SpargingStarted" )
      { S7_Templates := "time_type := Time" } "BatchTimer".Timer29.TON(pt := T#1S, et =>)
      R_Coil( "N2SpargingStarted" )
   END_RUNG
   RUNG wire#w1
      Contact( "N2SpargingPaused" )
      { S7_Templates := "time_type := Time" } "BatchTimer".Timer30.TON(pt := T#1S, et =>)
      R_Coil( "N2SpargingPaused" )
   END_RUNG
   RUNG wire#w1
      Contact( "N2SpargingResumed" )
      { S7_Templates := "time_type := Time" } "BatchTimer".Timer31.TON(pt := T#1S, et =>)
      R_Coil( "N2SpargingResumed" )
   END_RUNG
   RUNG wire#w1
      Contact( "N2SpargingOver" )
      { S7_Templates := "time_type := Time" } "BatchTimer".Timer32.TON(pt := T#1S, et =>)
      R_Coil( "N2SpargingOver" )
   END_RUNG
   RUNG wire#w1
      Contact( "N2SpargingReset" )
      { S7_Templates := "time_type := Time" } "BatchTimer".Timer33.TON(pt := T#1S, et =>)
      R_Coil( "N2SpargingReset" )
   END_RUNG
   // the same network as SCL:
   "BatchTimer".Timer29.TON(IN := "AlwaysTRUE" AND "N2SpargingStarted", PT := T#1S);
   IF "BatchTimer".Timer29.Q THEN "N2SpargingStarted" := FALSE; END_IF;
   "BatchTimer".Timer30.TON(IN := "AlwaysTRUE" AND "N2SpargingPaused", PT := T#1S);
   IF "BatchTimer".Timer30.Q THEN "N2SpargingPaused" := FALSE; END_IF;
   "BatchTimer".Timer31.TON(IN := "AlwaysTRUE" AND "N2SpargingResumed", PT := T#1S);
   IF "BatchTimer".Timer31.Q THEN "N2SpargingResumed" := FALSE; END_IF;
   "BatchTimer".Timer32.TON(IN := "AlwaysTRUE" AND "N2SpargingOver", PT := T#1S);
   IF "BatchTimer".Timer32.Q THEN "N2SpargingOver" := FALSE; END_IF;
   "BatchTimer".Timer33.TON(IN := "AlwaysTRUE" AND "N2SpargingReset", PT := T#1S);
   IF "BatchTimer".Timer33.Q THEN "N2SpargingReset" := FALSE; END_IF;
END_REGION

REGION Network 39: EventsResetTimer Gas Blanketing
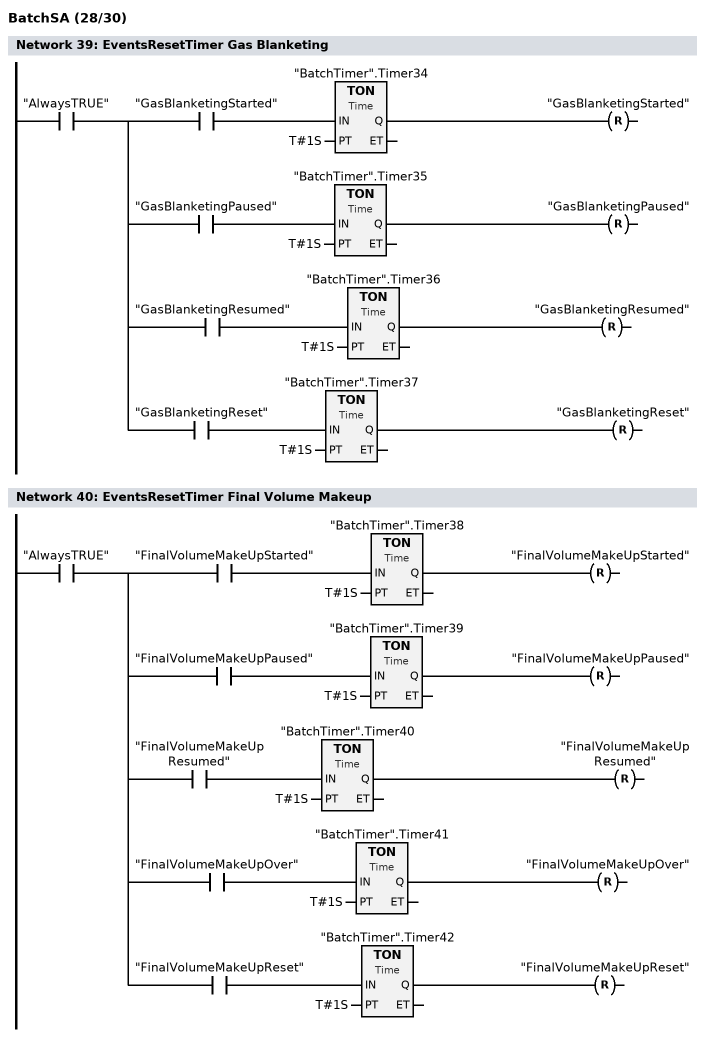
   RUNG wire#powerrail
      Contact( "AlwaysTRUE" )
      wire#w1
      Contact( "GasBlanketingStarted" )
      { S7_Templates := "time_type := Time" } "BatchTimer".Timer34.TON(pt := T#1S, et =>)
      R_Coil( "GasBlanketingStarted" )
   END_RUNG
   RUNG wire#w1
      Contact( "GasBlanketingPaused" )
      { S7_Templates := "time_type := Time" } "BatchTimer".Timer35.TON(pt := T#1S, et =>)
      R_Coil( "GasBlanketingPaused" )
   END_RUNG
   RUNG wire#w1
      Contact( "GasBlanketingResumed" )
      { S7_Templates := "time_type := Time" } "BatchTimer".Timer36.TON(pt := T#1S, et =>)
      R_Coil( "GasBlanketingResumed" )
   END_RUNG
   RUNG wire#w1
      Contact( "GasBlanketingReset" )
      { S7_Templates := "time_type := Time" } "BatchTimer".Timer37.TON(pt := T#1S, et =>)
      R_Coil( "GasBlanketingReset" )
   END_RUNG
   // the same network as SCL:
   "BatchTimer".Timer34.TON(IN := "AlwaysTRUE" AND "GasBlanketingStarted", PT := T#1S);
   IF "BatchTimer".Timer34.Q THEN "GasBlanketingStarted" := FALSE; END_IF;
   "BatchTimer".Timer35.TON(IN := "AlwaysTRUE" AND "GasBlanketingPaused", PT := T#1S);
   IF "BatchTimer".Timer35.Q THEN "GasBlanketingPaused" := FALSE; END_IF;
   "BatchTimer".Timer36.TON(IN := "AlwaysTRUE" AND "GasBlanketingResumed", PT := T#1S);
   IF "BatchTimer".Timer36.Q THEN "GasBlanketingResumed" := FALSE; END_IF;
   "BatchTimer".Timer37.TON(IN := "AlwaysTRUE" AND "GasBlanketingReset", PT := T#1S);
   IF "BatchTimer".Timer37.Q THEN "GasBlanketingReset" := FALSE; END_IF;
END_REGION

REGION Network 40: EventsResetTimer Final Volume Makeup
   RUNG wire#powerrail
      Contact( "AlwaysTRUE" )
      wire#w1
      Contact( "FinalVolumeMakeUpStarted" )
      { S7_Templates := "time_type := Time" } "BatchTimer".Timer38.TON(pt := T#1S, et =>)
      R_Coil( "FinalVolumeMakeUpStarted" )
   END_RUNG
   RUNG wire#w1
      Contact( "FinalVolumeMakeUpPaused" )
      { S7_Templates := "time_type := Time" } "BatchTimer".Timer39.TON(pt := T#1S, et =>)
      R_Coil( "FinalVolumeMakeUpPaused" )
   END_RUNG
   RUNG wire#w1
      Contact( "FinalVolumeMakeUpResumed" )
      { S7_Templates := "time_type := Time" } "BatchTimer".Timer40.TON(pt := T#1S, et =>)
      R_Coil( "FinalVolumeMakeUpResumed" )
   END_RUNG
   RUNG wire#w1
      Contact( "FinalVolumeMakeUpOver" )
      { S7_Templates := "time_type := Time" } "BatchTimer".Timer41.TON(pt := T#1S, et =>)
      R_Coil( "FinalVolumeMakeUpOver" )
   END_RUNG
   RUNG wire#w1
      Contact( "FinalVolumeMakeUpReset" )
      { S7_Templates := "time_type := Time" } "BatchTimer".Timer42.TON(pt := T#1S, et =>)
      R_Coil( "FinalVolumeMakeUpReset" )
   END_RUNG
   // the same network as SCL:
   "BatchTimer".Timer38.TON(IN := "AlwaysTRUE" AND "FinalVolumeMakeUpStarted", PT := T#1S);
   IF "BatchTimer".Timer38.Q THEN "FinalVolumeMakeUpStarted" := FALSE; END_IF;
   "BatchTimer".Timer39.TON(IN := "AlwaysTRUE" AND "FinalVolumeMakeUpPaused", PT := T#1S);
   IF "BatchTimer".Timer39.Q THEN "FinalVolumeMakeUpPaused" := FALSE; END_IF;
   "BatchTimer".Timer40.TON(IN := "AlwaysTRUE" AND "FinalVolumeMakeUpResumed", PT := T#1S);
   IF "BatchTimer".Timer40.Q THEN "FinalVolumeMakeUpResumed" := FALSE; END_IF;
   "BatchTimer".Timer41.TON(IN := "AlwaysTRUE" AND "FinalVolumeMakeUpOver", PT := T#1S);
   IF "BatchTimer".Timer41.Q THEN "FinalVolumeMakeUpOver" := FALSE; END_IF;
   "BatchTimer".Timer42.TON(IN := "AlwaysTRUE" AND "FinalVolumeMakeUpReset", PT := T#1S);
   IF "BatchTimer".Timer42.Q THEN "FinalVolumeMakeUpReset" := FALSE; END_IF;
END_REGION

REGION Network 41: EventsResetTimer Jacket
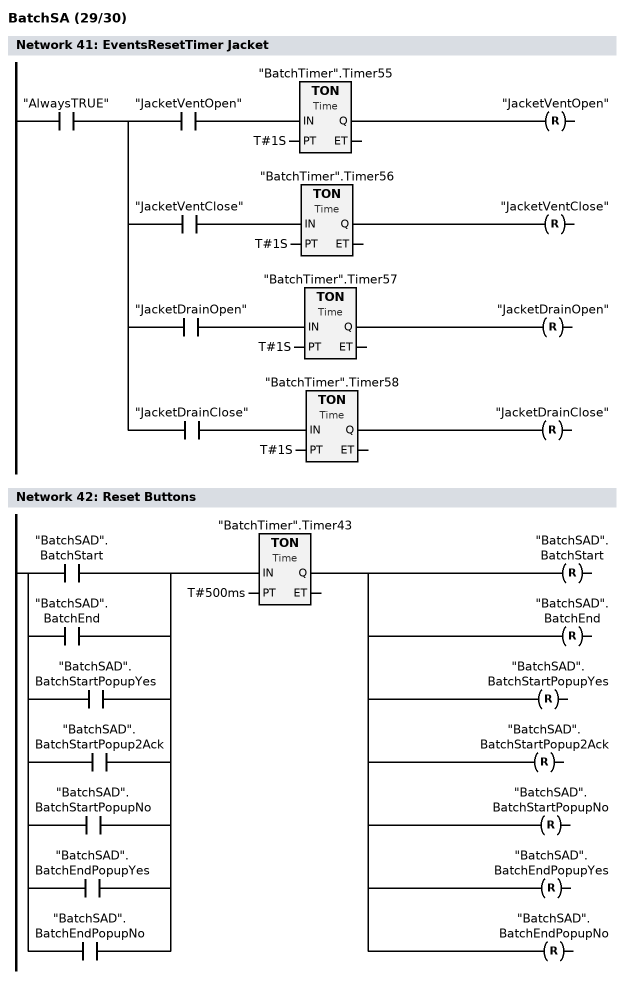
   RUNG wire#powerrail
      Contact( "AlwaysTRUE" )
      wire#w1
      Contact( "JacketVentOpen" )
      { S7_Templates := "time_type := Time" } "BatchTimer".Timer55.TON(pt := T#1S, et =>)
      R_Coil( "JacketVentOpen" )
   END_RUNG
   RUNG wire#w1
      Contact( "JacketVentClose" )
      { S7_Templates := "time_type := Time" } "BatchTimer".Timer56.TON(pt := T#1S, et =>)
      R_Coil( "JacketVentClose" )
   END_RUNG
   RUNG wire#w1
      Contact( "JacketDrainOpen" )
      { S7_Templates := "time_type := Time" } "BatchTimer".Timer57.TON(pt := T#1S, et =>)
      R_Coil( "JacketDrainOpen" )
   END_RUNG
   RUNG wire#w1
      Contact( "JacketDrainClose" )
      { S7_Templates := "time_type := Time" } "BatchTimer".Timer58.TON(pt := T#1S, et =>)
      R_Coil( "JacketDrainClose" )
   END_RUNG
   // the same network as SCL:
   "BatchTimer".Timer55.TON(IN := "AlwaysTRUE" AND "JacketVentOpen", PT := T#1S);
   IF "BatchTimer".Timer55.Q THEN "JacketVentOpen" := FALSE; END_IF;
   "BatchTimer".Timer56.TON(IN := "AlwaysTRUE" AND "JacketVentClose", PT := T#1S);
   IF "BatchTimer".Timer56.Q THEN "JacketVentClose" := FALSE; END_IF;
   "BatchTimer".Timer57.TON(IN := "AlwaysTRUE" AND "JacketDrainOpen", PT := T#1S);
   IF "BatchTimer".Timer57.Q THEN "JacketDrainOpen" := FALSE; END_IF;
   "BatchTimer".Timer58.TON(IN := "AlwaysTRUE" AND "JacketDrainClose", PT := T#1S);
   IF "BatchTimer".Timer58.Q THEN "JacketDrainClose" := FALSE; END_IF;
END_REGION

REGION Network 42: Reset Buttons
   RUNG wire#powerrail
      Contact( "BatchSAD".BatchStart )
      wire#w1
      { S7_Templates := "time_type := Time" } "BatchTimer".Timer43.TON(pt := T#500ms, et =>)
      wire#w2
      R_Coil( "BatchSAD".BatchStart )
   END_RUNG
   RUNG wire#powerrail
      Contact( "BatchSAD".BatchEnd )
   END_RUNG wire#w1
   RUNG wire#powerrail
      Contact( "BatchSAD".BatchStartPopupYes )
   END_RUNG wire#w1
   RUNG wire#powerrail
      Contact( "BatchSAD".BatchStartPopup2Ack )
   END_RUNG wire#w1
   RUNG wire#powerrail
      Contact( "BatchSAD".BatchStartPopupNo )
   END_RUNG wire#w1
   RUNG wire#powerrail
      Contact( "BatchSAD".BatchEndPopupYes )
   END_RUNG wire#w1
   RUNG wire#powerrail
      Contact( "BatchSAD".BatchEndPopupNo )
   END_RUNG wire#w1
   RUNG wire#w2
      R_Coil( "BatchSAD".BatchEnd )
   END_RUNG
   RUNG wire#w2
      R_Coil( "BatchSAD".BatchStartPopupYes )
   END_RUNG
   RUNG wire#w2
      R_Coil( "BatchSAD".BatchStartPopup2Ack )
   END_RUNG
   RUNG wire#w2
      R_Coil( "BatchSAD".BatchStartPopupNo )
   END_RUNG
   RUNG wire#w2
      R_Coil( "BatchSAD".BatchEndPopupYes )
   END_RUNG
   RUNG wire#w2
      R_Coil( "BatchSAD".BatchEndPopupNo )
   END_RUNG
   // the same network as SCL:
   "BatchTimer".Timer43.TON(IN := "BatchSAD".BatchStart OR "BatchSAD".BatchEnd OR "BatchSAD".BatchStartPopupYes OR "BatchSAD".BatchStartPopup2Ack OR "BatchSAD".BatchStartPopupNo OR "BatchSAD".BatchEndPopupYes OR "BatchSAD".BatchEndPopupNo,
                           PT := T#500ms);
   IF "BatchTimer".Timer43.Q THEN
       "BatchSAD".BatchStart := FALSE;
       "BatchSAD".BatchEnd := FALSE;
       "BatchSAD".BatchStartPopupYes := FALSE;
       "BatchSAD".BatchStartPopup2Ack := FALSE;
       "BatchSAD".BatchStartPopupNo := FALSE;
       "BatchSAD".BatchEndPopupYes := FALSE;
       "BatchSAD".BatchEndPopupNo := FALSE;
   END_IF;
END_REGION

REGION Network 43: RESET
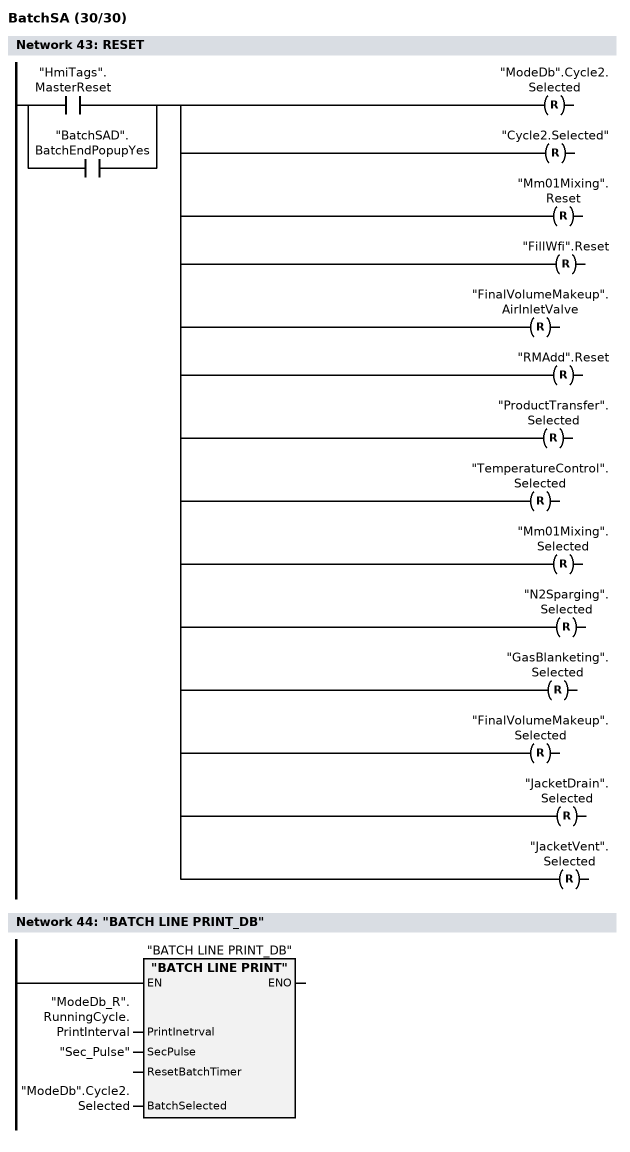
   RUNG wire#powerrail
      Contact( "HmiTags".MasterReset )
      wire#w1
      R_Coil( "ModeDb".Cycle2.Selected )
   END_RUNG
   RUNG wire#powerrail
      Contact( "BatchSAD".BatchEndPopupYes )
   END_RUNG wire#w1
   RUNG wire#w1
      R_Coil( "Cycle2.Selected" )
   END_RUNG
   RUNG wire#w1
      R_Coil( "Mm01Mixing".Reset )
   END_RUNG
   RUNG wire#w1
      R_Coil( "FillWfi".Reset )
   END_RUNG
   RUNG wire#w1
      R_Coil( "FinalVolumeMakeup".AirInletValve )
   END_RUNG
   RUNG wire#w1
      R_Coil( "RMAdd".Reset )
   END_RUNG
   RUNG wire#w1
      R_Coil( "ProductTransfer".Selected )
   END_RUNG
   RUNG wire#w1
      R_Coil( "TemperatureControl".Selected )
   END_RUNG
   RUNG wire#w1
      R_Coil( "Mm01Mixing".Selected )
   END_RUNG
   RUNG wire#w1
      R_Coil( "N2Sparging".Selected )
   END_RUNG
   RUNG wire#w1
      R_Coil( "GasBlanketing".Selected )
   END_RUNG
   RUNG wire#w1
      R_Coil( "FinalVolumeMakeup".Selected )
   END_RUNG
   RUNG wire#w1
      R_Coil( "JacketDrain".Selected )
   END_RUNG
   RUNG wire#w1
      R_Coil( "JacketVent".Selected )
   END_RUNG
   // the same network as SCL:
   IF "HmiTags".MasterReset OR "BatchSAD".BatchEndPopupYes THEN
       "ModeDb".Cycle2.Selected := FALSE;
       "Cycle2.Selected" := FALSE;
       "Mm01Mixing".Reset := FALSE;
       "FillWfi".Reset := FALSE;
       "FinalVolumeMakeup".AirInletValve := FALSE;
       "RMAdd".Reset := FALSE;
       "ProductTransfer".Selected := FALSE;
       "TemperatureControl".Selected := FALSE;
       "Mm01Mixing".Selected := FALSE;
       "N2Sparging".Selected := FALSE;
       "GasBlanketing".Selected := FALSE;
       "FinalVolumeMakeup".Selected := FALSE;
       "JacketDrain".Selected := FALSE;
       "JacketVent".Selected := FALSE;
   END_IF;
END_REGION

REGION Network 44: "BATCH LINE PRINT_DB"
   RUNG wire#powerrail
      "BATCH LINE PRINT_DB"(PrintInetrval := "ModeDb_R".RunningCycle.PrintInterval, SecPulse := "Sec_Pulse", ResetBatchTimer :=, BatchSelected := "ModeDb".Cycle2.Selected)
   END_RUNG
   // the same network as SCL:
   "BATCH LINE PRINT_DB"(PrintInetrval := "ModeDb_R".RunningCycle.PrintInterval,   // "BATCH LINE PRINT"
                         SecPulse := "Sec_Pulse",
                         BatchSelected := "ModeDb".Cycle2.Selected);
END_REGION
END_FUNCTION

FUNCTION_BLOCK "FB301"   // FB301, LAD
TITLE = FB301
{ S7_Optimized_Access := 'TRUE' }
AUTHOR : PRECISE
FAMILY : PRECISE
// FILLING/FINAL VOLUME MAKEUP
// stored: AutoNumber false, MemoryReserve 100, SetENOAutomatically false
   VAR_INPUT
      Enable : Bool;
      Disable : Bool;
      Fault : Bool;
      SecPulse : Bool;
      AlwaysTrue : Bool;
      StartConfirmationPopupSel : Bool;   // StartConfirmationPopupSel: 0-NO/1-YES
      EndConfirmationPopupSel : Bool;   // EndConfirmationPopupSel: 0-NO/1-YES
      FillModeSel : Int;   // Filling Mode Selection: 0-Auto/1-Manual
      FillMethodSel : Int;   // Filling Method Selection: 0-Weight/1-Time
      FillTimeBaseSel : Bool;   // Filling Time Base Selection: 0-second/1-minute
      FillLineSel : Int;   // Filling Line Selection: 0-J tube/1-SBI
      InitialDrainSel : Bool;
      SBIPulsingSel : Bool;
      FinalVolumeMakeupSel : Bool;
      PurgingSel : Bool;
      UtilitySel : Bool;   // Utility Selection: 0-PW/1-WFI
      FillQuantity : Real := 10.0;   // For Filling Method Slection: 0-Weight
      FillTimeMin : Int := 1;   // For Filling Method Slection: 1-Time
      FillTimeSec : Int := 30;   // For Filling Method Slection: 1-Time
      ActualQuantity : Real;   // For Filling Method Slection: 0-Weight
      InflightQuantity : Real;   // For Filling Method Slection: 0-Weight
      ZDVDelay : Int := 3;
      InitialDrainDelay : Int := 10;   // For Initial Drain Selection: Yes
      PurgingTime : Int := 10;   // For Purging Selection: Yes
      SBIOnTime : Int := 3;   // For SBI Pulsing Selection: Yes
      SBIOffTime : Int := 4;   // For SBI Pulsing Selection: Yes
      SetQuantitytoStartPulsing : Real := 10.0;   // For SBI Pulsing Selection: Yes
      FillQuantityTolerance : Real := 3.0;   // For Filling Method Slection: 0-Weight
      PrintInetrval : Int;
   END_VAR
   VAR_OUTPUT
      PWZDV : Bool;   // For Utility Selection: 0-PW
      WFIZDV : Bool;   // For Utility Selection: 1-WFI
      PWLineValves : Bool;   // For Utility Selection: 0-PW
      WFILineValves : Bool;   // For Utility Selection: 1-WFI
      InitialDrainValves : Bool;   // For Initial Drain Selection: Yes
      SBIValve : Bool;   // For Filling Line Selection: 1-SBI
      JTubeValve : Bool;   // For Filling Line Selection: 0-J tube
      AirInletValve : Bool;   // For Purging Selection: Yes
      StartConfirmationPopup : Bool;   // For Start Confirmation Popup Selection: Yes
      EndConfirmationPopup : Bool;   // For End Confirmation Popup Selection: Yes
      ManualPopup : Bool;   // For Filling Mode Selection: 1-Manual
      AlarmFillQuantityExeeded : Bool;
      FillTimeMinPV : DInt;   // For Filling Method Slection: 1-Time
      FillTimeSecPV : DInt;   // For Filling Method Slection: 1-Time
      PrintTrigger : Bool;
      PrintWord : Int;
      PrintStatus : String[50];
   END_VAR
   VAR_IN_OUT
      Start : Bool;
      Stop : Bool;
      Reset : Bool;
      StartConfirmationAck : Bool;   // For Start Confirmation Popup Selection: Yes
      EndConfirmationAck : Bool;   // For End Confirmation Popup Selection: Yes
      ManualAck : Bool;   // For Filling Mode Selection: 1-Manual
      AlarmAck : Bool;
      SpareBtn1 : Bool;
      Running : Bool;
      Selected : Bool;
      Paused : Bool;
      StartConfirmationPopupTemp : Bool;   // For Start Confirmation Popup Selection: Yes
      EndConfirmationPopupTemp : Bool;   // For End Confirmation Popup Selection: Yes
      ManualPopupTemp : Bool;   // For Filling Mode Selection: 1-Manual
      InitialDrainDelayStarted : Bool;
      InitialDrainDelayOver : Bool;
      FillStarted : Bool;
      FillOver : Bool;
      FillOverTemp : Bool;
      InitialDrainDelayPV : Int;
      ActualFillQuantityCalc : Real;   // For Filling Method Slection: 0-Weight
      ActualFillQuantity : Real;   // For Filling Method Slection: 0-Weight
      PulsingStartWeight : Real;   // For SBI Pulsing Selection: Yes
      PurgingTimePV : Int;   // For Purging Selection: Yes
      FillQuantityToleranceCalc : Real := 3.0;   // For Filling Method Slection: 0-Weight
      VesselMaxWeight : Real := 1000.0;
      ResetBatchTimer : Bool;
   END_VAR
   VAR
      ValveOnDelayPV : Int;
      ValveOffDelayPV : Int;
      PrintTriggerTemp : Bool;
      RE1 : Bool;
      RE2 : Bool;
      RE3 : Bool;
      RE4 : Bool;
      RE5 : Bool;
      RE6 : Bool;
      RE7 : Bool;
      FillTimer { S7_SetPoint := 'True'} : "FB101";
      SBIPulsing { S7_SetPoint := 'True'} : "FB102";
      PrintTriggerResetTimer { S7_SetPoint := 'True'} : TON_TIME;
      BtnResetTimer { S7_SetPoint := 'True'} : TON_TIME;
      IEC_Counter_0_Instance { S7_SetPoint := 'True'} : CTU_INT;
   END_VAR
   VAR_TEMP
      STATUS1 : String[40];
      STATUS2 : String[40];
      STATUS3 : String[40];
      STATUS4 : String[40];
      STATUS5 : String[40];
   END_VAR
   VAR_TEMP   // added for the SCL form of the ladder/FBD networks
      _w1 : Bool;
      _w2 : Bool;
      _w3 : Bool;
      _w4 : Bool;
      _w5 : Bool;
      _w6 : Bool;
   END_VAR
BEGIN

REGION Network 1: Running
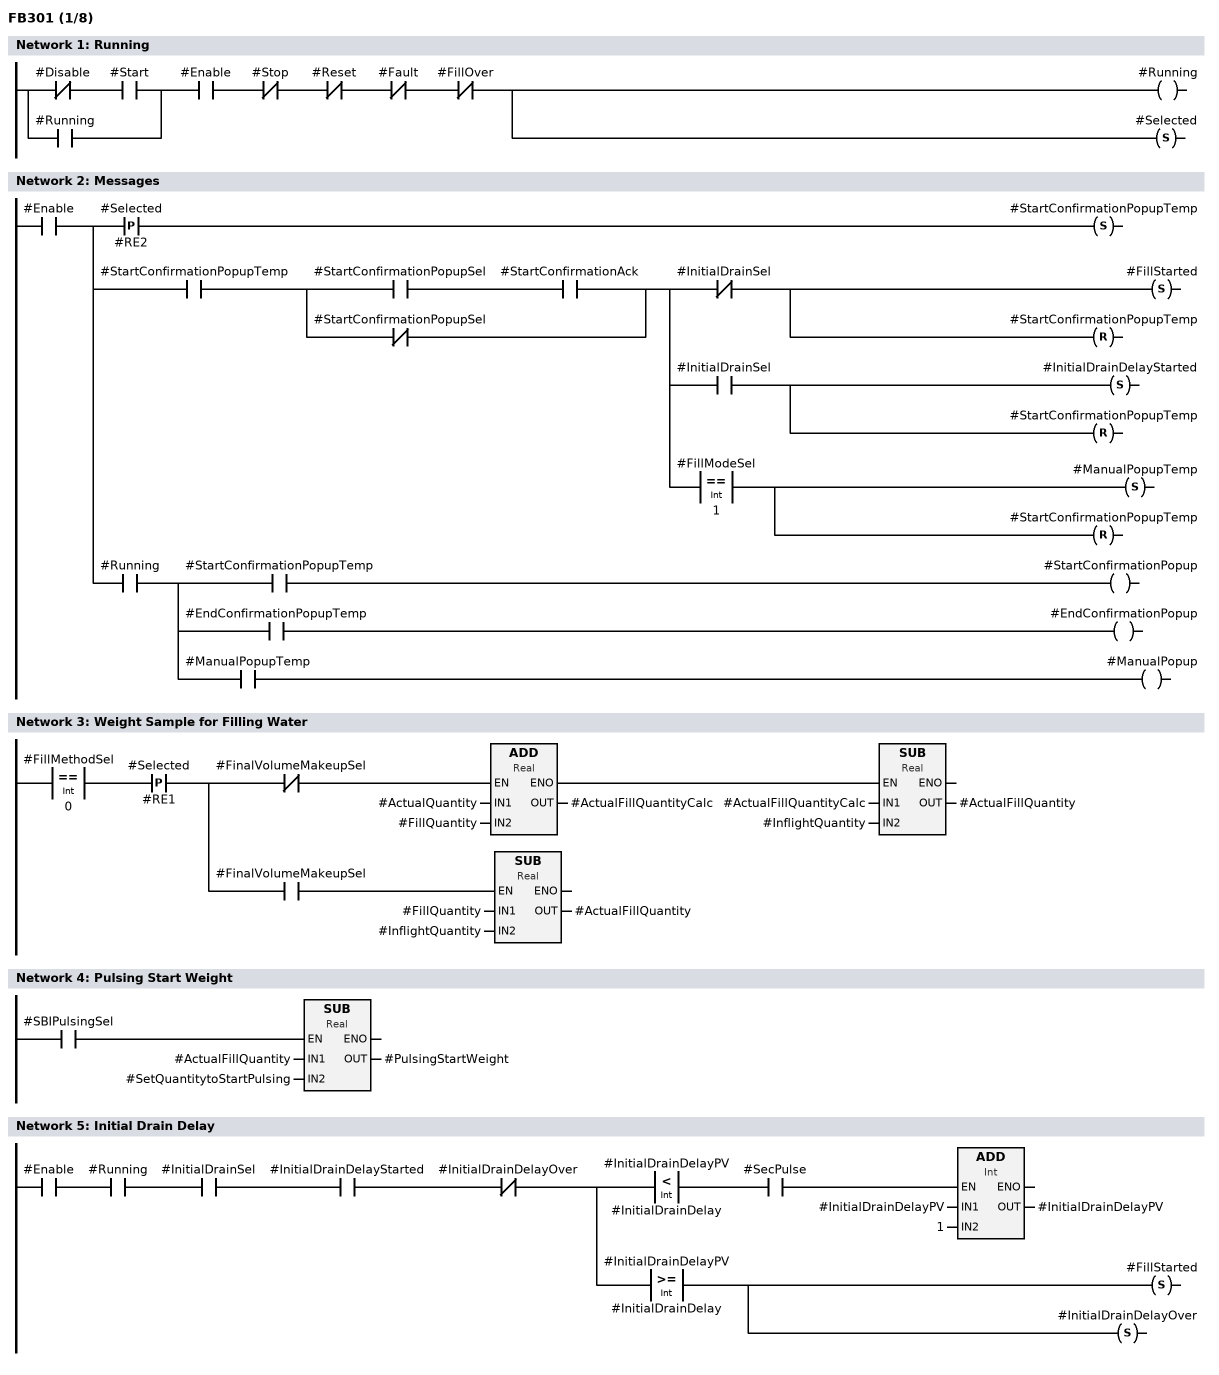
   RUNG wire#powerrail
      I_Contact( #Disable )
      Contact( #Start )
      wire#w1
      Contact( #Enable )
      I_Contact( #Stop )
      I_Contact( #Reset )
      I_Contact( #Fault )
      I_Contact( #FillOver )
      wire#w2
      Coil( #Running )
   END_RUNG
   RUNG wire#powerrail
      Contact( #Running )
   END_RUNG wire#w1
   RUNG wire#w2
      S_Coil( #Selected )
   END_RUNG
   // the same network as SCL:
   #Running := ((NOT #Disable AND #Start) OR #Running) AND #Enable AND NOT #Stop AND NOT #Reset AND NOT #Fault AND NOT #FillOver;
   IF #Running THEN #Selected := TRUE; END_IF;
END_REGION

REGION Network 2: Messages
   RUNG wire#powerrail
      Contact( #Enable )
      wire#w1
      P_Contact(operand := #Selected, bit := #RE2)
      S_Coil( #StartConfirmationPopupTemp )
   END_RUNG
   RUNG wire#w1
      Contact( #StartConfirmationPopupTemp )
      wire#w2
      Contact( #StartConfirmationPopupSel )
      Contact( #StartConfirmationAck )
      wire#w3
      I_Contact( #InitialDrainSel )
      wire#w4
      S_Coil( #FillStarted )
   END_RUNG
   RUNG wire#w2
      I_Contact( #StartConfirmationPopupSel )
   END_RUNG wire#w3
   RUNG wire#w4
      R_Coil( #StartConfirmationPopupTemp )
   END_RUNG
   RUNG wire#w3
      Contact( #InitialDrainSel )
      wire#w5
      S_Coil( #InitialDrainDelayStarted )
   END_RUNG
   RUNG wire#w5
      R_Coil( #StartConfirmationPopupTemp )
   END_RUNG
   RUNG wire#w3
      { S7_Templates := "SrcType := Int" } EQ_Contact(in1 := #FillModeSel, in2 := 1)
      wire#w6
      S_Coil( #ManualPopupTemp )
   END_RUNG
   RUNG wire#w6
      R_Coil( #StartConfirmationPopupTemp )
   END_RUNG
   RUNG wire#w1
      Contact( #Running )
      wire#w7
      Contact( #StartConfirmationPopupTemp )
      Coil( #StartConfirmationPopup )
   END_RUNG
   RUNG wire#w7
      Contact( #EndConfirmationPopupTemp )
      Coil( #EndConfirmationPopup )
   END_RUNG
   RUNG wire#w7
      Contact( #ManualPopupTemp )
      Coil( #ManualPopup )
   END_RUNG
   // the same network as SCL:
   #_w1 := #Enable AND #Selected AND NOT #RE2;   // rising edge of #Selected
   #RE2 := #Selected;
   IF #_w1 THEN #StartConfirmationPopupTemp := TRUE; END_IF;
   #_w2 := #Enable AND #StartConfirmationPopupTemp AND ((#StartConfirmationPopupSel AND #StartConfirmationAck) OR NOT #StartConfirmationPopupSel);
   IF #_w2 AND NOT #InitialDrainSel THEN
       #FillStarted := TRUE;
       #StartConfirmationPopupTemp := FALSE;
   END_IF;
   IF #_w2 AND #InitialDrainSel THEN
       #InitialDrainDelayStarted := TRUE;
       #StartConfirmationPopupTemp := FALSE;
   END_IF;
   IF #_w2 AND (#FillModeSel = 1) THEN
       #ManualPopupTemp := TRUE;
       #StartConfirmationPopupTemp := FALSE;
   END_IF;
   #_w3 := #Enable AND #Running;
   #StartConfirmationPopup := #_w3 AND #StartConfirmationPopupTemp;
   #EndConfirmationPopup := #_w3 AND #EndConfirmationPopupTemp;
   #ManualPopup := #_w3 AND #ManualPopupTemp;
END_REGION

REGION Network 3: Weight Sample for Filling Water
   RUNG wire#powerrail
      { S7_Templates := "SrcType := Int" } EQ_Contact(in1 := #FillMethodSel, in2 := 0)
      P_Contact(operand := #Selected, bit := #RE1)
      wire#w1
      I_Contact( #FinalVolumeMakeupSel )
      { S7_Templates := "SrcType := Real"; S7_GenerateENO := "TRUE" } Add(in1 := #ActualQuantity, in2 := #FillQuantity, out => #ActualFillQuantityCalc)
      { S7_Templates := "SrcType := Real"; S7_GenerateENO := "TRUE" } Sub(in1 := #ActualFillQuantityCalc, in2 := #InflightQuantity, out => #ActualFillQuantity)
   END_RUNG
   RUNG wire#w1
      Contact( #FinalVolumeMakeupSel )
      { S7_Templates := "SrcType := Real"; S7_GenerateENO := "TRUE" } Sub(in1 := #FillQuantity, in2 := #InflightQuantity, out => #ActualFillQuantity)
   END_RUNG
   // the same network as SCL:
   // ENO of a box is taken as its EN; it also drops when the box reports an error
   #_w1 := (#FillMethodSel = 0) AND #Selected AND NOT #RE1;   // rising edge of #Selected
   #RE1 := #Selected;
   IF #_w1 AND NOT #FinalVolumeMakeupSel THEN
       #ActualFillQuantityCalc := #ActualQuantity + #FillQuantity;
       #ActualFillQuantity := #ActualFillQuantityCalc - #InflightQuantity;
   END_IF;
   IF #_w1 AND #FinalVolumeMakeupSel THEN #ActualFillQuantity := #FillQuantity - #InflightQuantity; END_IF;
END_REGION

REGION Network 4: Pulsing Start Weight
   RUNG wire#powerrail
      Contact( #SBIPulsingSel )
      { S7_Templates := "SrcType := Real"; S7_GenerateENO := "TRUE" } Sub(in1 := #ActualFillQuantity, in2 := #SetQuantitytoStartPulsing, out => #PulsingStartWeight)
   END_RUNG
   // the same network as SCL:
   IF #SBIPulsingSel THEN #PulsingStartWeight := #ActualFillQuantity - #SetQuantitytoStartPulsing; END_IF;
END_REGION

REGION Network 5: Initial Drain Delay
   RUNG wire#powerrail
      Contact( #Enable )
      Contact( #Running )
      Contact( #InitialDrainSel )
      Contact( #InitialDrainDelayStarted )
      I_Contact( #InitialDrainDelayOver )
      wire#w1
      { S7_Templates := "SrcType := Int" } LT_Contact(in1 := #InitialDrainDelayPV, in2 := #InitialDrainDelay)
      Contact( #SecPulse )
      { S7_Templates := "SrcType := Int"; S7_GenerateENO := "TRUE" } Add(in1 := #InitialDrainDelayPV, in2 := 1, out => #InitialDrainDelayPV)
   END_RUNG
   RUNG wire#w1
      { S7_Templates := "SrcType := Int" } GE_Contact(in1 := #InitialDrainDelayPV, in2 := #InitialDrainDelay)
      wire#w2
      S_Coil( #FillStarted )
   END_RUNG
   RUNG wire#w2
      S_Coil( #InitialDrainDelayOver )
   END_RUNG
   // the same network as SCL:
   #_w1 := #Enable AND #Running AND #InitialDrainSel AND #InitialDrainDelayStarted AND NOT #InitialDrainDelayOver;
   IF #_w1 AND (#InitialDrainDelayPV < #InitialDrainDelay) AND #SecPulse THEN
       #InitialDrainDelayPV := #InitialDrainDelayPV + 1;
   END_IF;
   IF #_w1 AND (#InitialDrainDelayPV >= #InitialDrainDelay) THEN
       #FillStarted := TRUE;
       #InitialDrainDelayOver := TRUE;
   END_IF;
END_REGION

REGION Network 6: Fill Timer
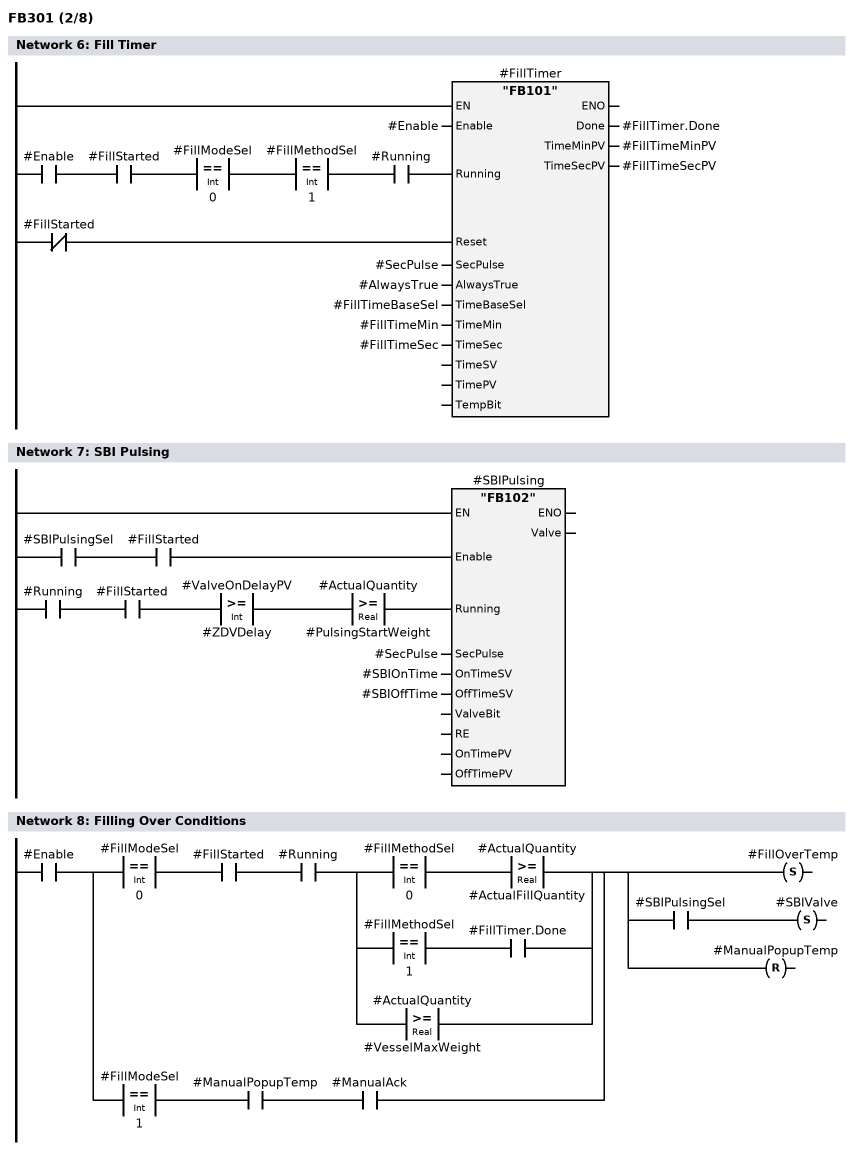
   RUNG wire#powerrail
      #FillTimer(Running := wire#w1, Reset := wire#w2, Enable := #Enable, SecPulse := #SecPulse, AlwaysTrue := #AlwaysTrue, TimeBaseSel := #FillTimeBaseSel, TimeMin := #FillTimeMin, TimeSec := #FillTimeSec, TimeSV :=, TimePV :=, TempBit :=, Done => #FillTimer.Done, TimeMinPV => #FillTimeMinPV, TimeSecPV => #FillTimeSecPV)
   END_RUNG
   RUNG wire#powerrail
      Contact( #Enable )
      Contact( #FillStarted )
      { S7_Templates := "SrcType := Int" } EQ_Contact(in1 := #FillModeSel, in2 := 0)
      { S7_Templates := "SrcType := Int" } EQ_Contact(in1 := #FillMethodSel, in2 := 1)
      Contact( #Running )
   END_RUNG wire#w1
   RUNG wire#powerrail
      I_Contact( #FillStarted )
   END_RUNG wire#w2
   // the same network as SCL:
   #FillTimer(Enable := #Enable,   // "FB101"
              Running := #Enable AND #FillStarted AND (#FillModeSel = 0) AND (#FillMethodSel = 1) AND #Running,
              Reset := NOT #FillStarted,
              SecPulse := #SecPulse,
              AlwaysTrue := #AlwaysTrue,
              TimeBaseSel := #FillTimeBaseSel,
              TimeMin := #FillTimeMin,
              TimeSec := #FillTimeSec,
              Done => #FillTimer.Done,
              TimeMinPV => #FillTimeMinPV,
              TimeSecPV => #FillTimeSecPV);
END_REGION

REGION Network 7: SBI Pulsing
   RUNG wire#powerrail
      #SBIPulsing(Enable := wire#w1, Running := wire#w2, SecPulse := #SecPulse, OnTimeSV := #SBIOnTime, OffTimeSV := #SBIOffTime, ValveBit :=, RE :=, OnTimePV :=, OffTimePV :=, Valve =>)
   END_RUNG
   RUNG wire#powerrail
      Contact( #SBIPulsingSel )
      Contact( #FillStarted )
   END_RUNG wire#w1
   RUNG wire#powerrail
      Contact( #Running )
      Contact( #FillStarted )
      { S7_Templates := "SrcType := Int" } GE_Contact(in1 := #ValveOnDelayPV, in2 := #ZDVDelay)
      { S7_Templates := "SrcType := Real" } GE_Contact(in1 := #ActualQuantity, in2 := #PulsingStartWeight)
   END_RUNG wire#w2
   // the same network as SCL:
   #SBIPulsing(Enable := #SBIPulsingSel AND #FillStarted,   // "FB102"
               Running := #Running AND #FillStarted AND (#ValveOnDelayPV >= #ZDVDelay) AND (#ActualQuantity >= #PulsingStartWeight),
               SecPulse := #SecPulse,
               OnTimeSV := #SBIOnTime,
               OffTimeSV := #SBIOffTime);
END_REGION

REGION Network 8: Filling Over Conditions
   RUNG wire#powerrail
      Contact( #Enable )
      wire#w1
      { S7_Templates := "SrcType := Int" } EQ_Contact(in1 := #FillModeSel, in2 := 0)
      Contact( #FillStarted )
      Contact( #Running )
      wire#w2
      { S7_Templates := "SrcType := Int" } EQ_Contact(in1 := #FillMethodSel, in2 := 0)
      { S7_Templates := "SrcType := Real" } GE_Contact(in1 := #ActualQuantity, in2 := #ActualFillQuantity)
      wire#w3
      S_Coil( #FillOverTemp )
   END_RUNG
   RUNG wire#w2
      { S7_Templates := "SrcType := Int" } EQ_Contact(in1 := #FillMethodSel, in2 := 1)
      Contact( #FillTimer.Done )
   END_RUNG wire#w3
   RUNG wire#w2
      { S7_Templates := "SrcType := Real" } GE_Contact(in1 := #ActualQuantity, in2 := #VesselMaxWeight)
   END_RUNG wire#w3
   RUNG wire#w1
      { S7_Templates := "SrcType := Int" } EQ_Contact(in1 := #FillModeSel, in2 := 1)
      Contact( #ManualPopupTemp )
      Contact( #ManualAck )
   END_RUNG wire#w3
   RUNG wire#w3
      Contact( #SBIPulsingSel )
      S_Coil( #SBIValve )
   END_RUNG
   RUNG wire#w3
      R_Coil( #ManualPopupTemp )
   END_RUNG
   // the same network as SCL:
   #_w1 := #Enable AND (((#FillModeSel = 0) AND #FillStarted AND #Running AND (((#FillMethodSel = 0) AND (#ActualQuantity >= #ActualFillQuantity)) OR ((#FillMethodSel = 1) AND #FillTimer.Done) OR (#ActualQuantity >= #VesselMaxWeight))) OR ((#FillModeSel = 1) AND #ManualPopupTemp AND #ManualAck));
   IF #_w1 THEN #FillOverTemp := TRUE; END_IF;
   IF #_w1 AND #SBIPulsingSel THEN #SBIValve := TRUE; END_IF;
   IF #_w1 THEN #ManualPopupTemp := FALSE; END_IF;
END_REGION

REGION Network 9: Purging Timer
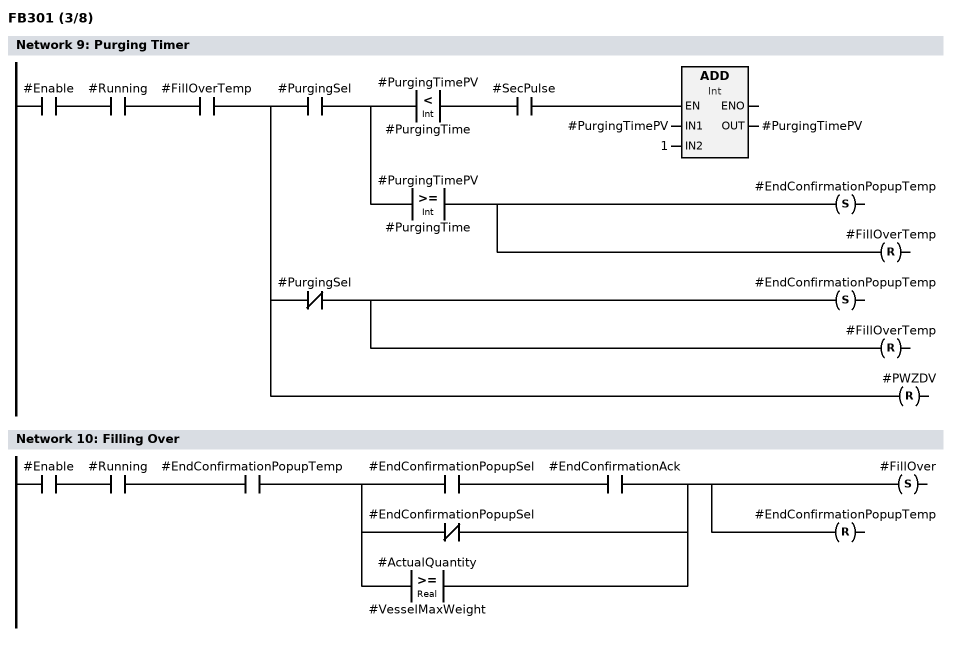
   RUNG wire#powerrail
      Contact( #Enable )
      Contact( #Running )
      Contact( #FillOverTemp )
      wire#w1
      Contact( #PurgingSel )
      wire#w2
      { S7_Templates := "SrcType := Int" } LT_Contact(in1 := #PurgingTimePV, in2 := #PurgingTime)
      Contact( #SecPulse )
      { S7_Templates := "SrcType := Int"; S7_GenerateENO := "TRUE" } Add(in1 := #PurgingTimePV, in2 := 1, out => #PurgingTimePV)
   END_RUNG
   RUNG wire#w2
      { S7_Templates := "SrcType := Int" } GE_Contact(in1 := #PurgingTimePV, in2 := #PurgingTime)
      wire#w3
      S_Coil( #EndConfirmationPopupTemp )
   END_RUNG
   RUNG wire#w3
      R_Coil( #FillOverTemp )
   END_RUNG
   RUNG wire#w1
      I_Contact( #PurgingSel )
      wire#w4
      S_Coil( #EndConfirmationPopupTemp )
   END_RUNG
   RUNG wire#w4
      R_Coil( #FillOverTemp )
   END_RUNG
   RUNG wire#w1
      R_Coil( #PWZDV )
   END_RUNG
   // the same network as SCL:
   #_w1 := #Enable AND #Running AND #FillOverTemp;
   #_w2 := #_w1 AND #PurgingSel;
   IF #_w2 AND (#PurgingTimePV < #PurgingTime) AND #SecPulse THEN
       #PurgingTimePV := #PurgingTimePV + 1;
   END_IF;
   IF #_w2 AND (#PurgingTimePV >= #PurgingTime) THEN
       #EndConfirmationPopupTemp := TRUE;
       #FillOverTemp := FALSE;
   END_IF;
   IF #_w1 AND NOT #PurgingSel THEN
       #EndConfirmationPopupTemp := TRUE;
       #FillOverTemp := FALSE;
   END_IF;
   IF #_w1 THEN #PWZDV := FALSE; END_IF;
END_REGION

REGION Network 10: Filling Over
   RUNG wire#powerrail
      Contact( #Enable )
      Contact( #Running )
      Contact( #EndConfirmationPopupTemp )
      wire#w1
      Contact( #EndConfirmationPopupSel )
      Contact( #EndConfirmationAck )
      wire#w2
      S_Coil( #FillOver )
   END_RUNG
   RUNG wire#w1
      I_Contact( #EndConfirmationPopupSel )
   END_RUNG wire#w2
   RUNG wire#w1
      { S7_Templates := "SrcType := Real" } GE_Contact(in1 := #ActualQuantity, in2 := #VesselMaxWeight)
   END_RUNG wire#w2
   RUNG wire#w2
      R_Coil( #EndConfirmationPopupTemp )
   END_RUNG
   // the same network as SCL:
   IF #Enable AND #Running AND #EndConfirmationPopupTemp AND ((#EndConfirmationPopupSel AND #EndConfirmationAck) OR NOT #EndConfirmationPopupSel OR (#ActualQuantity >= #VesselMaxWeight)) THEN
       #FillOver := TRUE;
       #EndConfirmationPopupTemp := FALSE;
   END_IF;
END_REGION

REGION Network 11: Output On
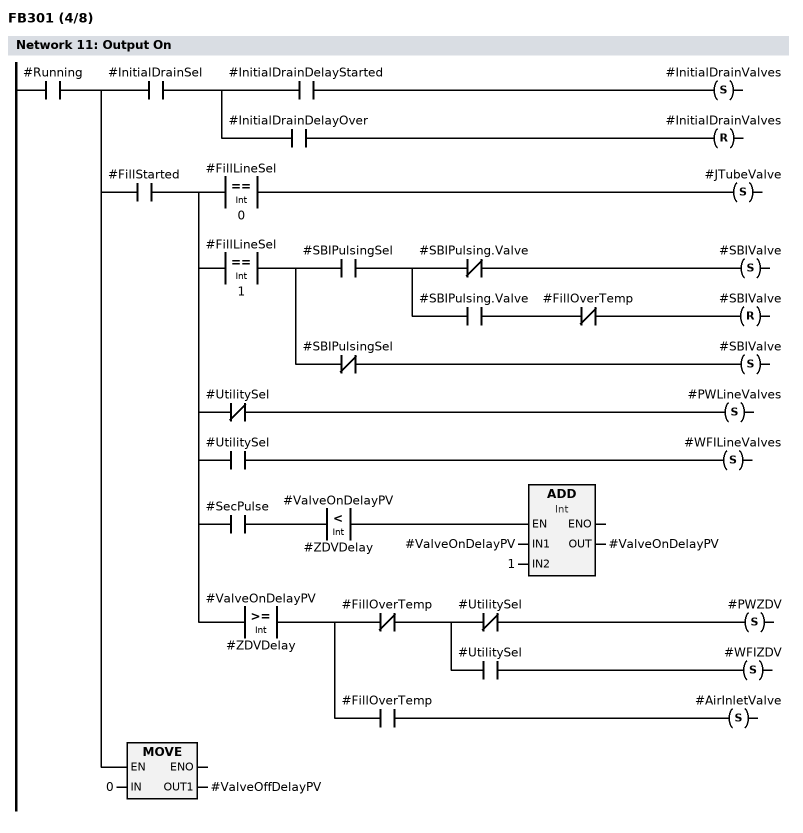
   RUNG wire#powerrail
      Contact( #Running )
      wire#w1
      Contact( #InitialDrainSel )
      wire#w2
      Contact( #InitialDrainDelayStarted )
      S_Coil( #InitialDrainValves )
   END_RUNG
   RUNG wire#w2
      Contact( #InitialDrainDelayOver )
      R_Coil( #InitialDrainValves )
   END_RUNG
   RUNG wire#w1
      Contact( #FillStarted )
      wire#w3
      { S7_Templates := "SrcType := Int" } EQ_Contact(in1 := #FillLineSel, in2 := 0)
      S_Coil( #JTubeValve )
   END_RUNG
   RUNG wire#w3
      { S7_Templates := "SrcType := Int" } EQ_Contact(in1 := #FillLineSel, in2 := 1)
      wire#w4
      Contact( #SBIPulsingSel )
      wire#w5
      I_Contact( #SBIPulsing.Valve )
      S_Coil( #SBIValve )
   END_RUNG
   RUNG wire#w5
      Contact( #SBIPulsing.Valve )
      I_Contact( #FillOverTemp )
      R_Coil( #SBIValve )
   END_RUNG
   RUNG wire#w4
      I_Contact( #SBIPulsingSel )
      S_Coil( #SBIValve )
   END_RUNG
   RUNG wire#w3
      I_Contact( #UtilitySel )
      S_Coil( #PWLineValves )
   END_RUNG
   RUNG wire#w3
      Contact( #UtilitySel )
      S_Coil( #WFILineValves )
   END_RUNG
   RUNG wire#w3
      Contact( #SecPulse )
      { S7_Templates := "SrcType := Int" } LT_Contact(in1 := #ValveOnDelayPV, in2 := #ZDVDelay)
      { S7_Templates := "SrcType := Int"; S7_GenerateENO := "TRUE" } Add(in1 := #ValveOnDelayPV, in2 := 1, out => #ValveOnDelayPV)
   END_RUNG
   RUNG wire#w3
      { S7_Templates := "SrcType := Int" } GE_Contact(in1 := #ValveOnDelayPV, in2 := #ZDVDelay)
      wire#w6
      I_Contact( #FillOverTemp )
      wire#w7
      I_Contact( #UtilitySel )
      S_Coil( #PWZDV )
   END_RUNG
   RUNG wire#w7
      Contact( #UtilitySel )
      S_Coil( #WFIZDV )
   END_RUNG
   RUNG wire#w6
      Contact( #FillOverTemp )
      S_Coil( #AirInletValve )
   END_RUNG
   RUNG wire#w1
      { S7_GenerateENO := "TRUE" } Move(in := 0, out1 => #ValveOffDelayPV)
   END_RUNG
   // the same network as SCL:
   #_w1 := #Running AND #InitialDrainSel;
   IF #_w1 AND #InitialDrainDelayStarted THEN #InitialDrainValves := TRUE; END_IF;
   IF #_w1 AND #InitialDrainDelayOver THEN #InitialDrainValves := FALSE; END_IF;
   #_w2 := #Running AND #FillStarted;
   IF #_w2 AND (#FillLineSel = 0) THEN #JTubeValve := TRUE; END_IF;
   #_w3 := #_w2 AND (#FillLineSel = 1);
   #_w4 := #_w3 AND #SBIPulsingSel;
   IF #_w4 AND NOT #SBIPulsing.Valve THEN #SBIValve := TRUE; END_IF;
   IF #_w4 AND #SBIPulsing.Valve AND NOT #FillOverTemp THEN #SBIValve := FALSE; END_IF;
   IF #_w3 AND NOT #SBIPulsingSel THEN #SBIValve := TRUE; END_IF;
   IF #_w2 AND NOT #UtilitySel THEN #PWLineValves := TRUE; END_IF;
   IF #_w2 AND #UtilitySel THEN #WFILineValves := TRUE; END_IF;
   IF #_w2 AND #SecPulse AND (#ValveOnDelayPV < #ZDVDelay) THEN
       #ValveOnDelayPV := #ValveOnDelayPV + 1;
   END_IF;
   #_w5 := #_w2 AND (#ValveOnDelayPV >= #ZDVDelay);
   #_w6 := #_w5 AND NOT #FillOverTemp;
   IF #_w6 AND NOT #UtilitySel THEN #PWZDV := TRUE; END_IF;
   IF #_w6 AND #UtilitySel THEN #WFIZDV := TRUE; END_IF;
   IF #_w5 AND #FillOverTemp THEN #AirInletValve := TRUE; END_IF;
   IF #Running THEN #ValveOffDelayPV := 0; END_IF;
END_REGION

REGION Network 12: Output Off
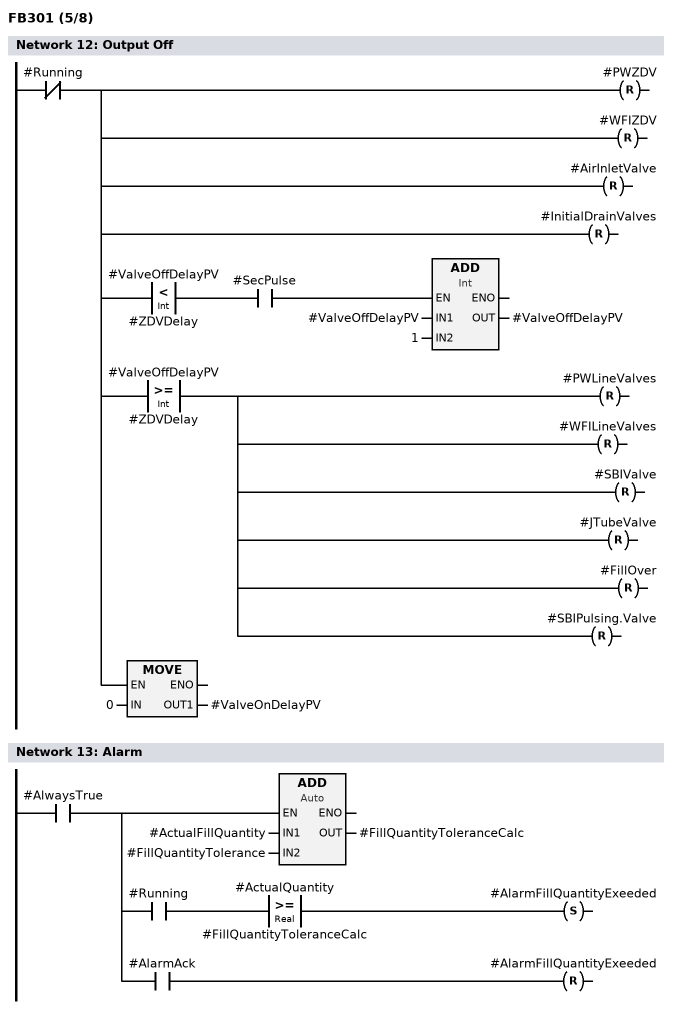
   RUNG wire#powerrail
      I_Contact( #Running )
      wire#w1
      R_Coil( #PWZDV )
   END_RUNG
   RUNG wire#w1
      R_Coil( #WFIZDV )
   END_RUNG
   RUNG wire#w1
      R_Coil( #AirInletValve )
   END_RUNG
   RUNG wire#w1
      R_Coil( #InitialDrainValves )
   END_RUNG
   RUNG wire#w1
      { S7_Templates := "SrcType := Int" } LT_Contact(in1 := #ValveOffDelayPV, in2 := #ZDVDelay)
      Contact( #SecPulse )
      { S7_Templates := "SrcType := Int"; S7_GenerateENO := "TRUE" } Add(in1 := #ValveOffDelayPV, in2 := 1, out => #ValveOffDelayPV)
   END_RUNG
   RUNG wire#w1
      { S7_Templates := "SrcType := Int" } GE_Contact(in1 := #ValveOffDelayPV, in2 := #ZDVDelay)
      wire#w2
      R_Coil( #PWLineValves )
   END_RUNG
   RUNG wire#w2
      R_Coil( #WFILineValves )
   END_RUNG
   RUNG wire#w2
      R_Coil( #SBIValve )
   END_RUNG
   RUNG wire#w2
      R_Coil( #JTubeValve )
   END_RUNG
   RUNG wire#w2
      R_Coil( #FillOver )
   END_RUNG
   RUNG wire#w2
      R_Coil( #SBIPulsing.Valve )
   END_RUNG
   RUNG wire#w1
      { S7_GenerateENO := "TRUE" } Move(in := 0, out1 => #ValveOnDelayPV)
   END_RUNG
   // the same network as SCL:
   IF NOT #Running THEN
       #PWZDV := FALSE;
       #WFIZDV := FALSE;
       #AirInletValve := FALSE;
       #InitialDrainValves := FALSE;
   END_IF;
   IF NOT #Running AND (#ValveOffDelayPV < #ZDVDelay) AND #SecPulse THEN
       #ValveOffDelayPV := #ValveOffDelayPV + 1;
   END_IF;
   IF NOT #Running AND (#ValveOffDelayPV >= #ZDVDelay) THEN
       #PWLineValves := FALSE;
       #WFILineValves := FALSE;
       #SBIValve := FALSE;
       #JTubeValve := FALSE;
       #FillOver := FALSE;
       #SBIPulsing.Valve := FALSE;
   END_IF;
   IF NOT #Running THEN #ValveOnDelayPV := 0; END_IF;
END_REGION

REGION Network 13: Alarm
   RUNG wire#powerrail
      Contact( #AlwaysTrue )
      wire#w1
      Add(in1 := #ActualFillQuantity, in2 := #FillQuantityTolerance, out => #FillQuantityToleranceCalc)
   END_RUNG
   RUNG wire#w1
      Contact( #Running )
      { S7_Templates := "SrcType := Real" } GE_Contact(in1 := #ActualQuantity, in2 := #FillQuantityToleranceCalc)
      S_Coil( #AlarmFillQuantityExeeded )
   END_RUNG
   RUNG wire#w1
      Contact( #AlarmAck )
      R_Coil( #AlarmFillQuantityExeeded )
   END_RUNG
   // the same network as SCL:
   IF #AlwaysTrue THEN #FillQuantityToleranceCalc := #ActualFillQuantity + #FillQuantityTolerance; END_IF;
   IF #AlwaysTrue AND #Running AND (#ActualQuantity >= #FillQuantityToleranceCalc) THEN
       #AlarmFillQuantityExeeded := TRUE;
   END_IF;
   IF #AlwaysTrue AND #AlarmAck THEN #AlarmFillQuantityExeeded := FALSE; END_IF;
END_REGION

REGION Network 14: Event Status
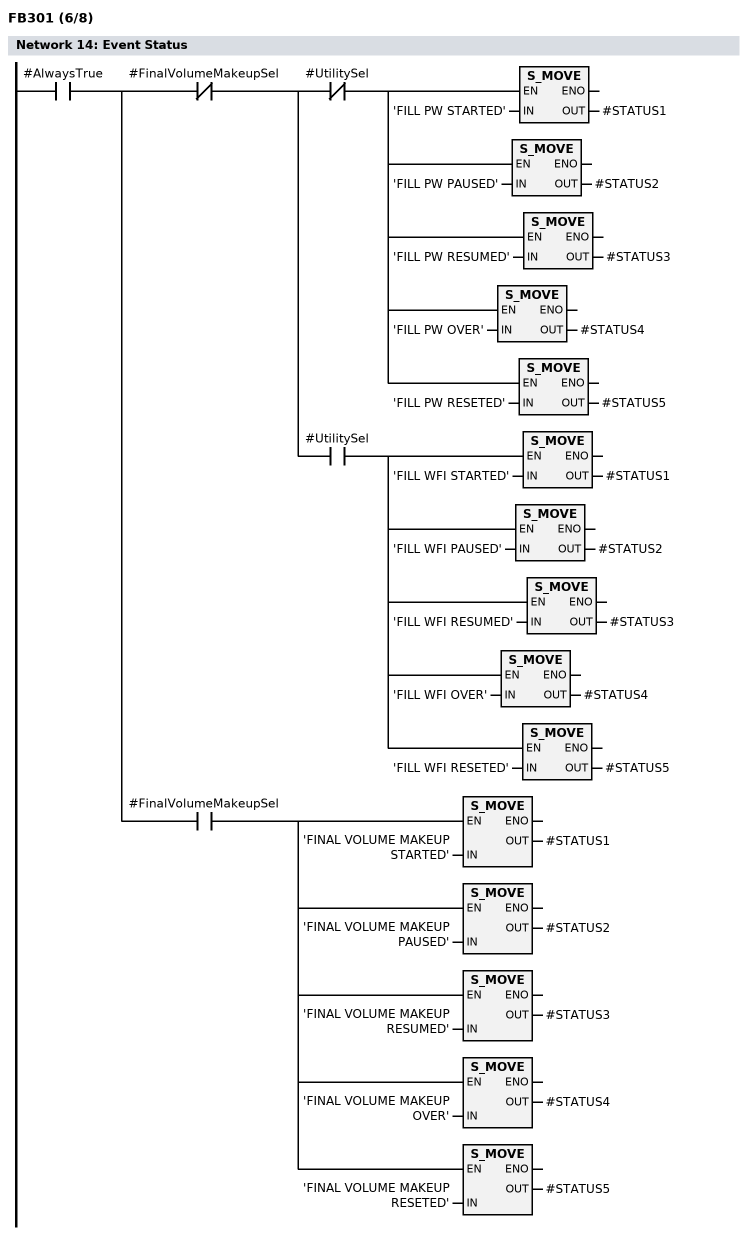
   RUNG wire#powerrail
      Contact( #AlwaysTrue )
      wire#w1
      I_Contact( #FinalVolumeMakeupSel )
      wire#w2
      I_Contact( #UtilitySel )
      wire#w3
      S_Move(in := 'FILL PW STARTED', out => #STATUS1)
   END_RUNG
   RUNG wire#w3
      S_Move(in := 'FILL PW PAUSED', out => #STATUS2)
   END_RUNG
   RUNG wire#w3
      S_Move(in := 'FILL PW RESUMED', out => #STATUS3)
   END_RUNG
   RUNG wire#w3
      S_Move(in := 'FILL PW OVER', out => #STATUS4)
   END_RUNG
   RUNG wire#w3
      S_Move(in := 'FILL PW RESETED', out => #STATUS5)
   END_RUNG
   RUNG wire#w2
      Contact( #UtilitySel )
      wire#w4
      S_Move(in := 'FILL WFI STARTED', out => #STATUS1)
   END_RUNG
   RUNG wire#w4
      S_Move(in := 'FILL WFI PAUSED', out => #STATUS2)
   END_RUNG
   RUNG wire#w4
      S_Move(in := 'FILL WFI RESUMED', out => #STATUS3)
   END_RUNG
   RUNG wire#w4
      S_Move(in := 'FILL WFI OVER', out => #STATUS4)
   END_RUNG
   RUNG wire#w4
      S_Move(in := 'FILL WFI RESETED', out => #STATUS5)
   END_RUNG
   RUNG wire#w1
      Contact( #FinalVolumeMakeupSel )
      wire#w5
      S_Move(in := 'FINAL VOLUME MAKEUP STARTED', out => #STATUS1)
   END_RUNG
   RUNG wire#w5
      S_Move(in := 'FINAL VOLUME MAKEUP PAUSED', out => #STATUS2)
   END_RUNG
   RUNG wire#w5
      S_Move(in := 'FINAL VOLUME MAKEUP RESUMED', out => #STATUS3)
   END_RUNG
   RUNG wire#w5
      S_Move(in := 'FINAL VOLUME MAKEUP OVER', out => #STATUS4)
   END_RUNG
   RUNG wire#w5
      S_Move(in := 'FINAL VOLUME MAKEUP RESETED', out => #STATUS5)
   END_RUNG
   // the same network as SCL:
   #_w1 := #AlwaysTrue AND NOT #FinalVolumeMakeupSel;
   IF #_w1 AND NOT #UtilitySel THEN
       #STATUS1 := 'FILL PW STARTED';
       #STATUS2 := 'FILL PW PAUSED';
       #STATUS3 := 'FILL PW RESUMED';
       #STATUS4 := 'FILL PW OVER';
       #STATUS5 := 'FILL PW RESETED';
   END_IF;
   IF #_w1 AND #UtilitySel THEN
       #STATUS1 := 'FILL WFI STARTED';
       #STATUS2 := 'FILL WFI PAUSED';
       #STATUS3 := 'FILL WFI RESUMED';
       #STATUS4 := 'FILL WFI OVER';
       #STATUS5 := 'FILL WFI RESETED';
   END_IF;
   IF #AlwaysTrue AND #FinalVolumeMakeupSel THEN
       #STATUS1 := 'FINAL VOLUME MAKEUP STARTED';
       #STATUS2 := 'FINAL VOLUME MAKEUP PAUSED';
       #STATUS3 := 'FINAL VOLUME MAKEUP RESUMED';
       #STATUS4 := 'FINAL VOLUME MAKEUP OVER';
       #STATUS5 := 'FINAL VOLUME MAKEUP RESETED';
   END_IF;
END_REGION

REGION Network 15: Print Logic
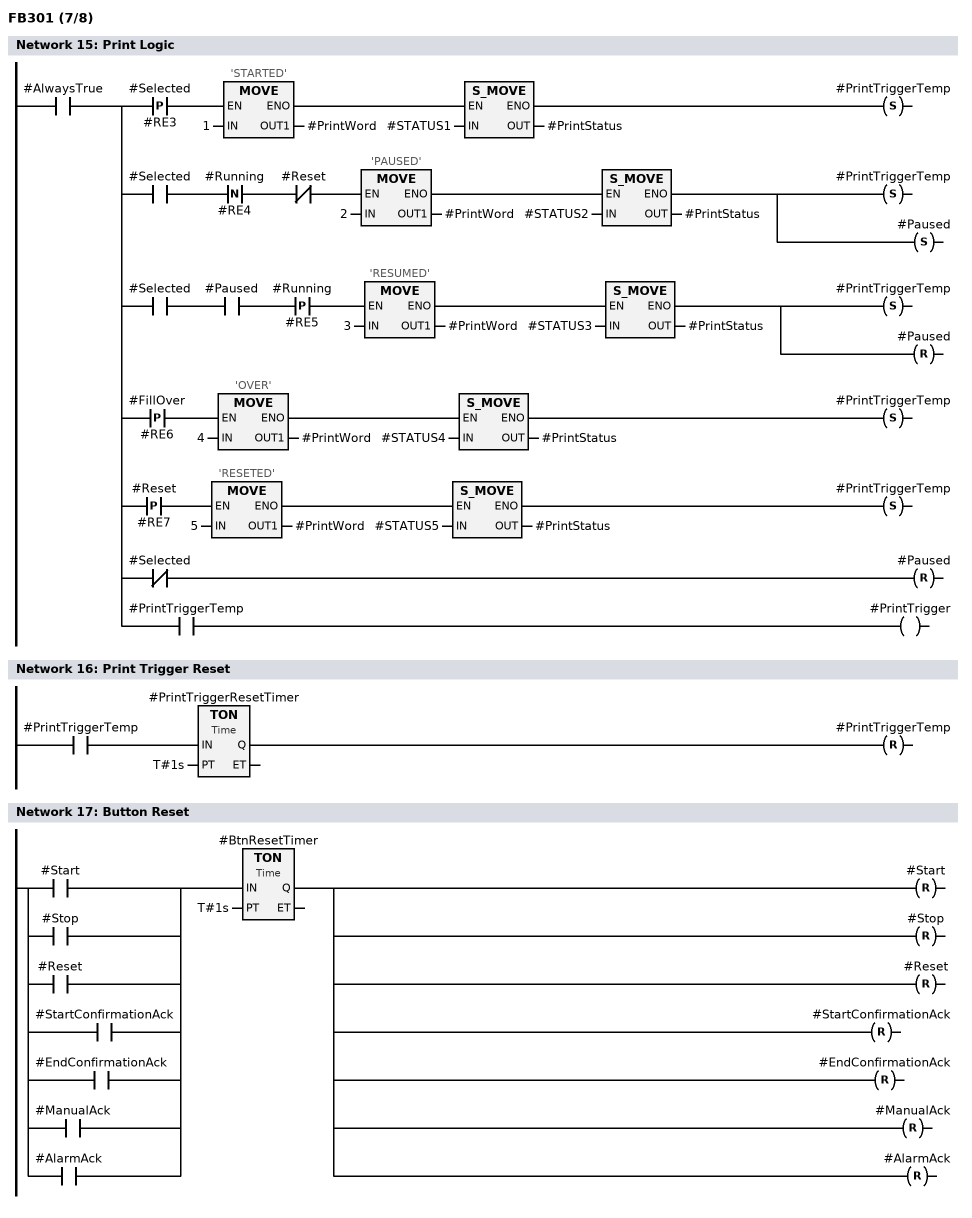
   RUNG wire#powerrail
      Contact( #AlwaysTrue )
      wire#w1
      P_Contact(operand := #Selected, bit := #RE3)
      { S7_GenerateENO := "TRUE" } Move(in := 1, out1 => #PrintWord)   // 'STARTED'
      S_Move(in := #STATUS1, out => #PrintStatus)
      S_Coil( #PrintTriggerTemp )
   END_RUNG
   RUNG wire#w1
      Contact( #Selected )
      N_Contact(operand := #Running, bit := #RE4)
      I_Contact( #Reset )
      { S7_GenerateENO := "TRUE" } Move(in := 2, out1 => #PrintWord)   // 'PAUSED'
      S_Move(in := #STATUS2, out => #PrintStatus)
      wire#w2
      S_Coil( #PrintTriggerTemp )
   END_RUNG
   RUNG wire#w2
      S_Coil( #Paused )
   END_RUNG
   RUNG wire#w1
      Contact( #Selected )
      Contact( #Paused )
      P_Contact(operand := #Running, bit := #RE5)
      { S7_GenerateENO := "TRUE" } Move(in := 3, out1 => #PrintWord)   // 'RESUMED'
      S_Move(in := #STATUS3, out => #PrintStatus)
      wire#w3
      S_Coil( #PrintTriggerTemp )
   END_RUNG
   RUNG wire#w3
      R_Coil( #Paused )
   END_RUNG
   RUNG wire#w1
      P_Contact(operand := #FillOver, bit := #RE6)
      { S7_GenerateENO := "TRUE" } Move(in := 4, out1 => #PrintWord)   // 'OVER'
      S_Move(in := #STATUS4, out => #PrintStatus)
      S_Coil( #PrintTriggerTemp )
   END_RUNG
   RUNG wire#w1
      P_Contact(operand := #Reset, bit := #RE7)
      { S7_GenerateENO := "TRUE" } Move(in := 5, out1 => #PrintWord)   // 'RESETED'
      S_Move(in := #STATUS5, out => #PrintStatus)
      S_Coil( #PrintTriggerTemp )
   END_RUNG
   RUNG wire#w1
      I_Contact( #Selected )
      R_Coil( #Paused )
   END_RUNG
   RUNG wire#w1
      Contact( #PrintTriggerTemp )
      Coil( #PrintTrigger )
   END_RUNG
   // the same network as SCL:
   // ENO of a box is taken as its EN; it also drops when the box reports an error
   #_w1 := #AlwaysTrue AND #Selected AND NOT #RE3;   // rising edge of #Selected
   #RE3 := #Selected;
   IF #_w1 THEN
       #PrintWord := 1;   // 'STARTED'
       #PrintStatus := #STATUS1;
       #PrintTriggerTemp := TRUE;
   END_IF;
   #_w2 := #AlwaysTrue AND #Selected AND NOT #Running AND #RE4;   // falling edge of #Running
   #RE4 := #Running;
   IF #_w2 AND NOT #Reset THEN
       #PrintWord := 2;   // 'PAUSED'
       #PrintStatus := #STATUS2;
       #PrintTriggerTemp := TRUE;
       #Paused := TRUE;
   END_IF;
   #_w3 := #AlwaysTrue AND #Selected AND #Paused AND #Running AND NOT #RE5;   // rising edge of #Running
   #RE5 := #Running;
   IF #_w3 THEN
       #PrintWord := 3;   // 'RESUMED'
       #PrintStatus := #STATUS3;
       #PrintTriggerTemp := TRUE;
       #Paused := FALSE;
   END_IF;
   #_w4 := #AlwaysTrue AND #FillOver AND NOT #RE6;   // rising edge of #FillOver
   #RE6 := #FillOver;
   IF #_w4 THEN
       #PrintWord := 4;   // 'OVER'
       #PrintStatus := #STATUS4;
       #PrintTriggerTemp := TRUE;
   END_IF;
   #_w5 := #AlwaysTrue AND #Reset AND NOT #RE7;   // rising edge of #Reset
   #RE7 := #Reset;
   IF #_w5 THEN
       #PrintWord := 5;   // 'RESETED'
       #PrintStatus := #STATUS5;
       #PrintTriggerTemp := TRUE;
   END_IF;
   IF #AlwaysTrue AND NOT #Selected THEN #Paused := FALSE; END_IF;
   #PrintTrigger := #AlwaysTrue AND #PrintTriggerTemp;
END_REGION

REGION Network 16: Print Trigger Reset
   RUNG wire#powerrail
      Contact( #PrintTriggerTemp )
      { S7_Templates := "time_type := Time" } #PrintTriggerResetTimer.TON(pt := T#1s, et =>)
      R_Coil( #PrintTriggerTemp )
   END_RUNG
   // the same network as SCL:
   #PrintTriggerResetTimer(IN := #PrintTriggerTemp, PT := T#1s);   // TON
   IF #PrintTriggerResetTimer.Q THEN #PrintTriggerTemp := FALSE; END_IF;
END_REGION

REGION Network 17: Button Reset
   RUNG wire#powerrail
      Contact( #Start )
      wire#w1
      { S7_Templates := "time_type := Time" } #BtnResetTimer.TON(pt := T#1s, et =>)
      wire#w2
      R_Coil( #Start )
   END_RUNG
   RUNG wire#powerrail
      Contact( #Stop )
   END_RUNG wire#w1
   RUNG wire#powerrail
      Contact( #Reset )
   END_RUNG wire#w1
   RUNG wire#powerrail
      Contact( #StartConfirmationAck )
   END_RUNG wire#w1
   RUNG wire#powerrail
      Contact( #EndConfirmationAck )
   END_RUNG wire#w1
   RUNG wire#powerrail
      Contact( #ManualAck )
   END_RUNG wire#w1
   RUNG wire#powerrail
      Contact( #AlarmAck )
   END_RUNG wire#w1
   RUNG wire#w2
      R_Coil( #Stop )
   END_RUNG
   RUNG wire#w2
      R_Coil( #Reset )
   END_RUNG
   RUNG wire#w2
      R_Coil( #StartConfirmationAck )
   END_RUNG
   RUNG wire#w2
      R_Coil( #EndConfirmationAck )
   END_RUNG
   RUNG wire#w2
      R_Coil( #ManualAck )
   END_RUNG
   RUNG wire#w2
      R_Coil( #AlarmAck )
   END_RUNG
   // the same network as SCL:
   #BtnResetTimer(IN := #Start OR #Stop OR #Reset OR #StartConfirmationAck OR #EndConfirmationAck OR #ManualAck OR #AlarmAck,   // TON
                  PT := T#1s);
   IF #BtnResetTimer.Q THEN
       #Start := FALSE;
       #Stop := FALSE;
       #Reset := FALSE;
       #StartConfirmationAck := FALSE;
       #EndConfirmationAck := FALSE;
       #ManualAck := FALSE;
       #AlarmAck := FALSE;
   END_IF;
END_REGION

REGION Network 18: Reset
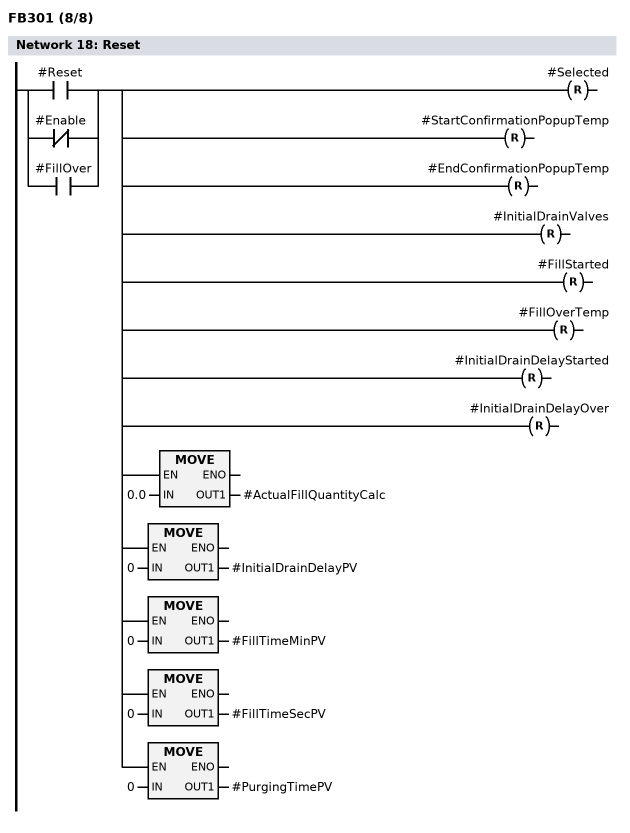
   RUNG wire#powerrail
      Contact( #Reset )
      wire#w1
      R_Coil( #Selected )
   END_RUNG
   RUNG wire#powerrail
      I_Contact( #Enable )
   END_RUNG wire#w1
   RUNG wire#powerrail
      Contact( #FillOver )
   END_RUNG wire#w1
   RUNG wire#w1
      R_Coil( #StartConfirmationPopupTemp )
   END_RUNG
   RUNG wire#w1
      R_Coil( #EndConfirmationPopupTemp )
   END_RUNG
   RUNG wire#w1
      R_Coil( #InitialDrainValves )
   END_RUNG
   RUNG wire#w1
      R_Coil( #FillStarted )
   END_RUNG
   RUNG wire#w1
      R_Coil( #FillOverTemp )
   END_RUNG
   RUNG wire#w1
      R_Coil( #InitialDrainDelayStarted )
   END_RUNG
   RUNG wire#w1
      R_Coil( #InitialDrainDelayOver )
   END_RUNG
   RUNG wire#w1
      { S7_GenerateENO := "TRUE" } Move(in := 0.0, out1 => #ActualFillQuantityCalc)
   END_RUNG
   RUNG wire#w1
      { S7_GenerateENO := "TRUE" } Move(in := 0, out1 => #InitialDrainDelayPV)
   END_RUNG
   RUNG wire#w1
      { S7_GenerateENO := "TRUE" } Move(in := 0, out1 => #FillTimeMinPV)
   END_RUNG
   RUNG wire#w1
      { S7_GenerateENO := "TRUE" } Move(in := 0, out1 => #FillTimeSecPV)
   END_RUNG
   RUNG wire#w1
      { S7_GenerateENO := "TRUE" } Move(in := 0, out1 => #PurgingTimePV)
   END_RUNG
   // the same network as SCL:
   IF #Reset OR NOT #Enable OR #FillOver THEN
       #Selected := FALSE;
       #StartConfirmationPopupTemp := FALSE;
       #EndConfirmationPopupTemp := FALSE;
       #InitialDrainValves := FALSE;
       #FillStarted := FALSE;
       #FillOverTemp := FALSE;
       #InitialDrainDelayStarted := FALSE;
       #InitialDrainDelayOver := FALSE;
       #ActualFillQuantityCalc := 0.0;
       #InitialDrainDelayPV := 0;
       #FillTimeMinPV := 0;
       #FillTimeSecPV := 0;
       #PurgingTimePV := 0;
   END_IF;
END_REGION
END_FUNCTION_BLOCK

FUNCTION_BLOCK "FB101"   // FB101, LAD
TITLE = FB101
{ S7_Optimized_Access := 'TRUE' }
AUTHOR : PRECISE
FAMILY : PRECISE
// TIMER (RETENTIVE)
// stored: AutoNumber false, MemoryReserve 100, SetENOAutomatically false
   VAR_INPUT
      Enable : Bool;
      Running : Bool;
      Reset : Bool;
      SecPulse : Bool;
      AlwaysTrue : Bool;
      TimeBaseSel : Bool;   // Time Base Selection: 0-second/1-minute
      TimeMin : Int;
      TimeSec : Int;
   END_VAR
   VAR_OUTPUT
      Done : Bool;
      TimeMinPV : DInt;
      TimeSecPV : DInt;
   END_VAR
   VAR_IN_OUT
      TimeSV : DInt;
      TimePV : DInt;
      TempBit : Bool;
   END_VAR
BEGIN

REGION Network 1: Set Time Min/Sec
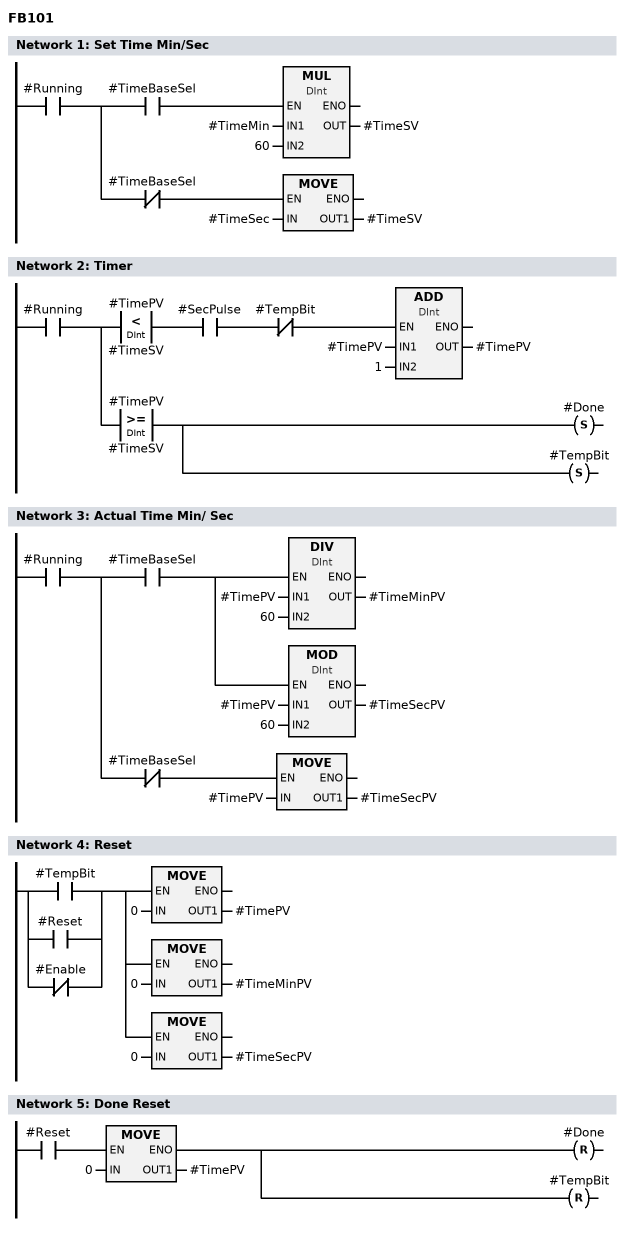
   RUNG wire#powerrail
      Contact( #Running )
      wire#w1
      Contact( #TimeBaseSel )
      { S7_Templates := "SrcType := DInt"; S7_GenerateENO := "TRUE" } Mul(in1 := #TimeMin, in2 := 60, out => #TimeSV)
   END_RUNG
   RUNG wire#w1
      I_Contact( #TimeBaseSel )
      { S7_GenerateENO := "TRUE" } Move(in := #TimeSec, out1 => #TimeSV)
   END_RUNG
   // the same network as SCL:
   IF #Running AND #TimeBaseSel THEN #TimeSV := #TimeMin * 60; END_IF;
   IF #Running AND NOT #TimeBaseSel THEN #TimeSV := #TimeSec; END_IF;
END_REGION

REGION Network 2: Timer
   RUNG wire#powerrail
      Contact( #Running )
      wire#w1
      { S7_Templates := "SrcType := DInt" } LT_Contact(in1 := #TimePV, in2 := #TimeSV)
      Contact( #SecPulse )
      I_Contact( #TempBit )
      { S7_Templates := "SrcType := DInt"; S7_GenerateENO := "TRUE" } Add(in1 := #TimePV, in2 := 1, out => #TimePV)
   END_RUNG
   RUNG wire#w1
      { S7_Templates := "SrcType := DInt" } GE_Contact(in1 := #TimePV, in2 := #TimeSV)
      wire#w2
      S_Coil( #Done )
   END_RUNG
   RUNG wire#w2
      S_Coil( #TempBit )
   END_RUNG
   // the same network as SCL:
   IF #Running AND (#TimePV < #TimeSV) AND #SecPulse AND NOT #TempBit THEN #TimePV := #TimePV + 1; END_IF;
   IF #Running AND (#TimePV >= #TimeSV) THEN
       #Done := TRUE;
       #TempBit := TRUE;
   END_IF;
END_REGION

REGION Network 3: Actual Time Min/ Sec
   RUNG wire#powerrail
      Contact( #Running )
      wire#w1
      Contact( #TimeBaseSel )
      wire#w2
      { S7_Templates := "SrcType := DInt"; S7_GenerateENO := "TRUE" } Div(in1 := #TimePV, in2 := 60, out => #TimeMinPV)
   END_RUNG
   RUNG wire#w2
      { S7_Templates := "SrcType := DInt"; S7_GenerateENO := "TRUE" } Mod(in1 := #TimePV, in2 := 60, out => #TimeSecPV)
   END_RUNG
   RUNG wire#w1
      I_Contact( #TimeBaseSel )
      { S7_GenerateENO := "TRUE" } Move(in := #TimePV, out1 => #TimeSecPV)
   END_RUNG
   // the same network as SCL:
   IF #Running AND #TimeBaseSel THEN
       #TimeMinPV := #TimePV / 60;
       #TimeSecPV := #TimePV MOD 60;
   END_IF;
   IF #Running AND NOT #TimeBaseSel THEN #TimeSecPV := #TimePV; END_IF;
END_REGION

REGION Network 4: Reset
   RUNG wire#powerrail
      Contact( #TempBit )
      wire#w1
      { S7_GenerateENO := "TRUE" } Move(in := 0, out1 => #TimePV)
   END_RUNG
   RUNG wire#powerrail
      Contact( #Reset )
   END_RUNG wire#w1
   RUNG wire#powerrail
      I_Contact( #Enable )
   END_RUNG wire#w1
   RUNG wire#w1
      { S7_GenerateENO := "TRUE" } Move(in := 0, out1 => #TimeMinPV)
   END_RUNG
   RUNG wire#w1
      { S7_GenerateENO := "TRUE" } Move(in := 0, out1 => #TimeSecPV)
   END_RUNG
   // the same network as SCL:
   IF #TempBit OR #Reset OR NOT #Enable THEN
       #TimePV := 0;
       #TimeMinPV := 0;
       #TimeSecPV := 0;
   END_IF;
END_REGION

REGION Network 5: Done Reset
   RUNG wire#powerrail
      Contact( #Reset )
      { S7_GenerateENO := "TRUE" } Move(in := 0, out1 => #TimePV)
      wire#w1
      R_Coil( #Done )
   END_RUNG
   RUNG wire#w1
      R_Coil( #TempBit )
   END_RUNG
   // the same network as SCL:
   // ENO of a box is taken as its EN; it also drops when the box reports an error
   IF #Reset THEN
       #TimePV := 0;
       #Done := FALSE;
       #TempBit := FALSE;
   END_IF;
END_REGION
END_FUNCTION_BLOCK

FUNCTION_BLOCK "FB102"   // FB102, LAD
TITLE = FB102
{ S7_Optimized_Access := 'FALSE' }
AUTHOR : PRECISE
FAMILY : PRECISE
// On Off Delay
// stored: AutoNumber false, SetENOAutomatically false
   VAR_INPUT
      Enable : Bool;
      Running : Bool;
      SecPulse : Bool;
      OnTimeSV : Int := 3;
      OffTimeSV : Int := 3;
   END_VAR
   VAR_OUTPUT
      Valve : Bool;
   END_VAR
   VAR_IN_OUT
      ValveBit : Bool;
      RE : Bool;
      OnTimePV : Int;
      OffTimePV : Int;
   END_VAR
   VAR_TEMP   // added for the SCL form of the ladder/FBD networks
      _w1 : Bool;
      _w2 : Bool;
      _w3 : Bool;
   END_VAR
BEGIN

REGION Network 1: Start
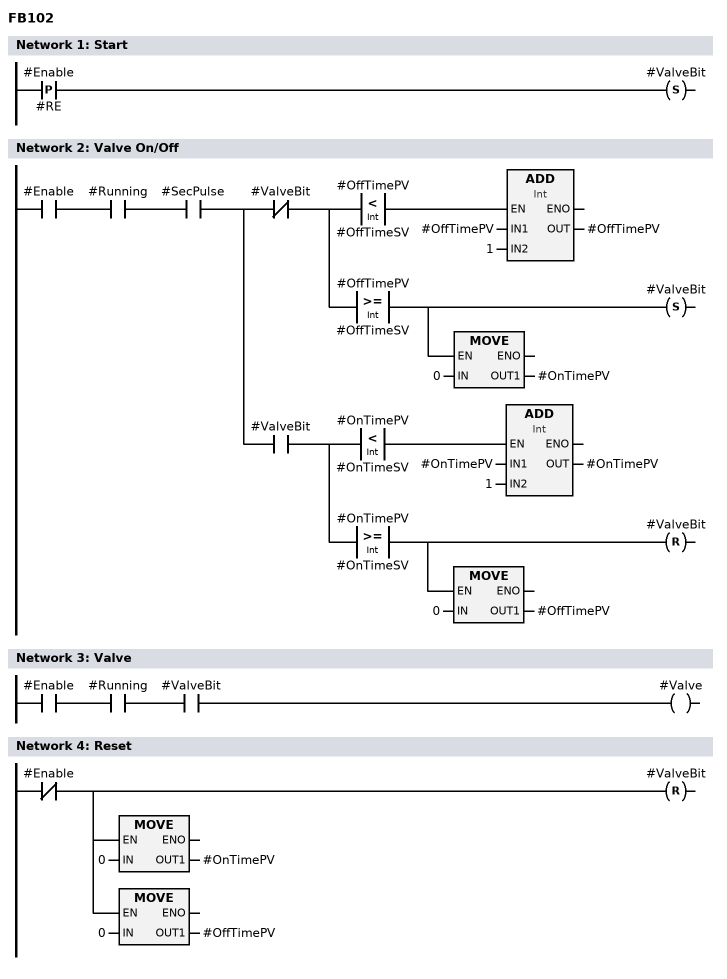
   RUNG wire#powerrail
      P_Contact(operand := #Enable, bit := #RE)
      S_Coil( #ValveBit )
   END_RUNG
   // the same network as SCL:
   #_w1 := #Enable AND NOT #RE;   // rising edge of #Enable
   #RE := #Enable;
   IF #_w1 THEN #ValveBit := TRUE; END_IF;
END_REGION

REGION Network 2: Valve On/Off
   RUNG wire#powerrail
      Contact( #Enable )
      Contact( #Running )
      Contact( #SecPulse )
      wire#w1
      I_Contact( #ValveBit )
      wire#w2
      { S7_Templates := "SrcType := Int" } LT_Contact(in1 := #OffTimePV, in2 := #OffTimeSV)
      { S7_Templates := "SrcType := Int"; S7_GenerateENO := "TRUE" } Add(in1 := #OffTimePV, in2 := 1, out => #OffTimePV)
   END_RUNG
   RUNG wire#w2
      { S7_Templates := "SrcType := Int" } GE_Contact(in1 := #OffTimePV, in2 := #OffTimeSV)
      wire#w3
      S_Coil( #ValveBit )
   END_RUNG
   RUNG wire#w3
      { S7_GenerateENO := "TRUE" } Move(in := 0, out1 => #OnTimePV)
   END_RUNG
   RUNG wire#w1
      Contact( #ValveBit )
      wire#w4
      { S7_Templates := "SrcType := Int" } LT_Contact(in1 := #OnTimePV, in2 := #OnTimeSV)
      { S7_Templates := "SrcType := Int"; S7_GenerateENO := "TRUE" } Add(in1 := #OnTimePV, in2 := 1, out => #OnTimePV)
   END_RUNG
   RUNG wire#w4
      { S7_Templates := "SrcType := Int" } GE_Contact(in1 := #OnTimePV, in2 := #OnTimeSV)
      wire#w5
      R_Coil( #ValveBit )
   END_RUNG
   RUNG wire#w5
      { S7_GenerateENO := "TRUE" } Move(in := 0, out1 => #OffTimePV)
   END_RUNG
   // the same network as SCL:
   #_w1 := #Enable AND #Running AND #SecPulse;
   #_w2 := #_w1 AND NOT #ValveBit;
   IF #_w2 AND (#OffTimePV < #OffTimeSV) THEN #OffTimePV := #OffTimePV + 1; END_IF;
   IF #_w2 AND (#OffTimePV >= #OffTimeSV) THEN
       #ValveBit := TRUE;
       #OnTimePV := 0;
   END_IF;
   #_w3 := #_w1 AND #ValveBit;
   IF #_w3 AND (#OnTimePV < #OnTimeSV) THEN #OnTimePV := #OnTimePV + 1; END_IF;
   IF #_w3 AND (#OnTimePV >= #OnTimeSV) THEN
       #ValveBit := FALSE;
       #OffTimePV := 0;
   END_IF;
END_REGION

REGION Network 3: Valve
   RUNG wire#powerrail
      Contact( #Enable )
      Contact( #Running )
      Contact( #ValveBit )
      Coil( #Valve )
   END_RUNG
   // the same network as SCL:
   #Valve := #Enable AND #Running AND #ValveBit;
END_REGION

REGION Network 4: Reset
   RUNG wire#powerrail
      I_Contact( #Enable )
      wire#w1
      R_Coil( #ValveBit )
   END_RUNG
   RUNG wire#w1
      { S7_GenerateENO := "TRUE" } Move(in := 0, out1 => #OnTimePV)
   END_RUNG
   RUNG wire#w1
      { S7_GenerateENO := "TRUE" } Move(in := 0, out1 => #OffTimePV)
   END_RUNG
   // the same network as SCL:
   IF NOT #Enable THEN
       #ValveBit := FALSE;
       #OnTimePV := 0;
       #OffTimePV := 0;
   END_IF;
END_REGION
END_FUNCTION_BLOCK

FUNCTION_BLOCK "FB311"   // FB311, LAD
TITLE = FB311
{ S7_Optimized_Access := 'TRUE' }
AUTHOR : PRECISE
FAMILY : PRECISE
// TEMPERATURE CONTROL
// stored: AutoNumber false, MemoryReserve 100, SetENOAutomatically false
   VAR_INPUT
      Enable : Bool;
      Disable : Bool;
      Fault : Bool;
      SecPulse : Bool;
      AlwaysTrue : Bool;
      StartConfirmationPopupSel : Bool;   // StartConfirmationPopupSel: 0-NO/1-YES
      EndConfirmationPopupSel : Bool;   // EndConfirmationPopupSel: 0-NO/1-YES
      TimebaseSel : Bool;   // Timebase Selection: 0-sec/1-min
      TemperatureMaintainSel : Bool;   // Temperature Maintain Selection: 0-NO/1-YES
      BypassSel : Bool;   // Bypass Selection: 0-NO/1-YES
      JacketAirPurgingSel : Bool;   // Applicable for if Air Inlet Valve is present in jacket. 0-NO/1-YES
      TemperatureControlSel : Int;   // Temperature Control Sel : 0-Heat/1-Cool
      SensorSel : Int;   // Sensor Slection: 0-Vessel/1-Jacket
      BatchSizeSel : Int;   // Batch Size Sel:0-Small/1-Big
      HeatingUtilitySel : Int;   // Heating Utility Selection: 0-Steam/1-Hot Water
      CoolingUtilitySelection : Int;   // 0-cooling/1-chilling/2-brine/3-cooling+chilling/4-chilling+brine/5-cooling+chilling+Brine
      SetTemperature : Real := 60.0;
      TimeMin : Int := 1;   // For Temperature Maintain Selection: 1-YES & Bypass Selection: 1-YES
      TimeSec : Int := 30;   // For Temperature Maintain Selection: 1-YES & Bypass Selection: 0-NO
      ActualTemperatureVessel : Real;   // For Sensor Slection: 0-Vessel
      ActualTemperatureJacket : Real;   // For Sensor Slection: 1-Jacket
      JVDelay : Int := 5;
      JDDelay : Int := 5;
      TemperatureTol : Real := 0.3;
      CoolingThreshold : Real := 25.0;   // Temperature to change utility from cooling water to chilled water
      ChillingThreshold : Real := 15.0;   // Temperature to change utility from chilled water to brine water
      HeatHighTemperatureTol : Real := 3.0;
      CoolLowTemperatureTol : Real := 3.0;
      JacketAirPurgingTimeSec : Int := 10;
   END_VAR
   VAR_OUTPUT
      JacketAirValve : Bool;
      BypassValve : Bool;
      JacketVentValve1 : Bool;
      JacketDrainValve1 : Bool;
      CoolingWaterInletValve1 : Bool;
      CoolingWaterOutletValve1 : Bool;
      ChilledWaterInletValve1 : Bool;
      ChilledWaterOutletValve1 : Bool;
      BrineWaterInletValve1 : Bool;
      BrineWaterOutletValve1 : Bool;
      HotWaterInletValve1 : Bool;
      HotWaterOutletValve1 : Bool;
      SteamInlet1 : Bool;
      Condensateoutlet1 : Bool;
      JacketVentValve2 : Bool;
      JacketDrainValve2 : Bool;
      CoolingWaterInletValve2 : Bool;
      CoolingWaterOutletValve2 : Bool;
      ChilledWaterInletValve2 : Bool;
      ChilledWaterOutletValve2 : Bool;
      BrineWaterInletValve2 : Bool;
      BrineWaterOutletValve2 : Bool;
      HotWaterInletValve2 : Bool;
      HotWaterOutletValve2 : Bool;
      SteamInlet2 : Bool;
      Condensateoutlet2 : Bool;
      AlarmHeatHighTemperature : Bool;
      AlarmCoolLowTemperature : Bool;
      StartConfirmationPopup : Bool;   // For Start Confirmation Popup Selection: Yes
      EndConfirmationPopup : Bool;   // For End Confirmation Popup Selection: Yes
      JacketAirPurgingPopup : Bool;
      TimeMinPV : DInt;
      TimeSecPV : DInt;
      JacketAirPurgingTimeSecPV : Int;
      PrintTrigger : Bool;
      PrintWord : Int;
      PrintStatus : String[50];
   END_VAR
   VAR_IN_OUT
      Start : Bool;
      Stop : Bool;
      Reset : Bool;
      StartConfirmationAck : Bool;   // For Start Confirmation Popup Selection: Yes
      EndConfirmationAck : Bool;   // For End Confirmation Popup Selection: Yes
      JacketAirPurgingAck : Bool;
      AlarmAck : Bool;
      SpareBtn1 : Bool;
      Running : Bool;
      Selected : Bool;
      Paused : Bool;
      StartConfirmationPopupTemp : Bool;   // For Start Confirmation Popup Selection: Yes
      EndConfirmationPopupTemp : Bool;   // For End Confirmation Popup Selection: Yes
      Started : Bool;
      Over : Bool;
      StartJVDelay : Bool;
      StartJDDelay : Bool;
      StartUtility : Bool;
      StartChilling : Bool;
      StartBrine : Bool;
      StartJacketAirPurging : Bool;
      HeatTempReached : Bool;
      CoolTempReached : Bool;
      TemperatureTolNeg : Real;
      TemperatureTolPos : Real;
      HeatHighTemperatureTolCal : Real := 3.0;
      CoolLowTemperatureTolCal : Real := 3.0;
      JacketPressureSelection : Bool;   // 0-no,1-yes
      JacketPressureReached : Bool;
      JacketUtilityPressureValve : Bool;
      JAcketAlarms : Bool;
      Temp : Bool;
      JacketTime : Int;
      JacketSafetyPressure : Real;
      JAcketActPressure : Real;
   END_VAR
   VAR
      PrintTriggerTemp : Bool;
      RE1 : Bool;
      RE2 : Bool;
      RE3 : Bool;
      RE4 : Bool;
      RE5 : Bool;
      RE6 : Bool;
      RE7 : Bool;
      RE8 : Bool;
      RE9 : Bool;
      RE10 : Bool;
      RE11 : Bool;
      "Timer" : "FB101";
      PrintTriggerResetTimer { S7_SetPoint := 'True'} : TON_TIME;
      BtnResetTimer { S7_SetPoint := 'True'} : TON_TIME;
      JVDelayTime { S7_SetPoint := 'True'} : "FB103";
      JDDelayTime { S7_SetPoint := 'True'} : "FB103";
      JAPTime { S7_SetPoint := 'True'} : "FB103";
      ActualTemperature : Real;
      JacketpressureTimer { S7_SetPoint := 'True'} : "FB103";
      FB101_Instance { S7_SetPoint := 'True'} : "FB101";
   END_VAR
   VAR_TEMP
      STATUS1 : String[40];
      STATUS2 : String[40];
      STATUS3 : String[40];
      STATUS4 : String[40];
      STATUS5 : String[40];
      STATUS6 : String[40];
   END_VAR
   VAR_TEMP   // added for the SCL form of the ladder/FBD networks
      _w1 : Bool;
      _w2 : Bool;
      _w3 : Bool;
      _w4 : Bool;
      _w5 : Bool;
      _w6 : Bool;
      _w7 : Bool;
      _w8 : Bool;
   END_VAR
BEGIN

REGION Network 1: Running
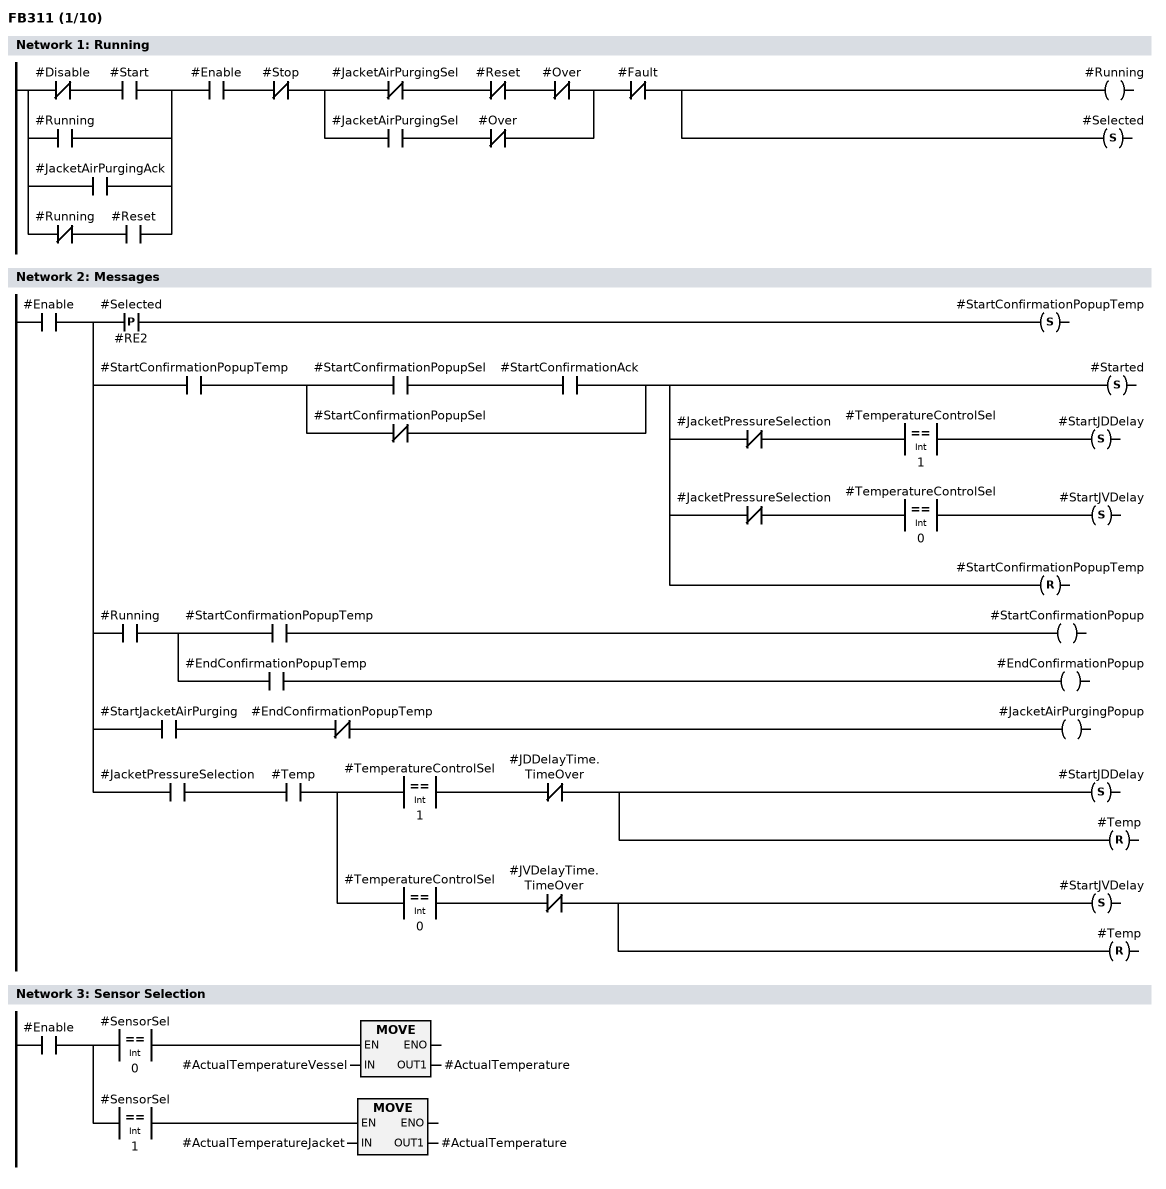
   RUNG wire#powerrail
      I_Contact( #Disable )
      Contact( #Start )
      wire#w1
      Contact( #Enable )
      I_Contact( #Stop )
      wire#w2
      I_Contact( #JacketAirPurgingSel )
      I_Contact( #Reset )
      I_Contact( #Over )
      wire#w3
      I_Contact( #Fault )
      wire#w4
      Coil( #Running )
   END_RUNG
   RUNG wire#powerrail
      Contact( #Running )
   END_RUNG wire#w1
   RUNG wire#powerrail
      Contact( #JacketAirPurgingAck )
   END_RUNG wire#w1
   RUNG wire#powerrail
      I_Contact( #Running )
      Contact( #Reset )
   END_RUNG wire#w1
   RUNG wire#w2
      Contact( #JacketAirPurgingSel )
      I_Contact( #Over )
   END_RUNG wire#w3
   RUNG wire#w4
      S_Coil( #Selected )
   END_RUNG
   // the same network as SCL:
   #Running := ((NOT #Disable AND #Start) OR #Running OR #JacketAirPurgingAck OR (NOT #Running AND #Reset)) AND #Enable AND NOT #Stop AND ((NOT #JacketAirPurgingSel AND NOT #Reset AND NOT #Over) OR (#JacketAirPurgingSel AND NOT #Over)) AND NOT #Fault;
   IF #Running THEN #Selected := TRUE; END_IF;
END_REGION

REGION Network 2: Messages
   RUNG wire#powerrail
      Contact( #Enable )
      wire#w1
      P_Contact(operand := #Selected, bit := #RE2)
      S_Coil( #StartConfirmationPopupTemp )
   END_RUNG
   RUNG wire#w1
      Contact( #StartConfirmationPopupTemp )
      wire#w2
      Contact( #StartConfirmationPopupSel )
      Contact( #StartConfirmationAck )
      wire#w3
      S_Coil( #Started )
   END_RUNG
   RUNG wire#w2
      I_Contact( #StartConfirmationPopupSel )
   END_RUNG wire#w3
   RUNG wire#w3
      I_Contact( #JacketPressureSelection )
      { S7_Templates := "SrcType := Int" } EQ_Contact(in1 := #TemperatureControlSel, in2 := 1)
      S_Coil( #StartJDDelay )
   END_RUNG
   RUNG wire#w3
      I_Contact( #JacketPressureSelection )
      { S7_Templates := "SrcType := Int" } EQ_Contact(in1 := #TemperatureControlSel, in2 := 0)
      S_Coil( #StartJVDelay )
   END_RUNG
   RUNG wire#w3
      R_Coil( #StartConfirmationPopupTemp )
   END_RUNG
   RUNG wire#w1
      Contact( #Running )
      wire#w4
      Contact( #StartConfirmationPopupTemp )
      Coil( #StartConfirmationPopup )
   END_RUNG
   RUNG wire#w4
      Contact( #EndConfirmationPopupTemp )
      Coil( #EndConfirmationPopup )
   END_RUNG
   RUNG wire#w1
      Contact( #StartJacketAirPurging )
      I_Contact( #EndConfirmationPopupTemp )
      Coil( #JacketAirPurgingPopup )
   END_RUNG
   RUNG wire#w1
      Contact( #JacketPressureSelection )
      Contact( #Temp )
      wire#w5
      { S7_Templates := "SrcType := Int" } EQ_Contact(in1 := #TemperatureControlSel, in2 := 1)
      I_Contact( #JDDelayTime.TimeOver )
      wire#w6
      S_Coil( #StartJDDelay )
   END_RUNG
   RUNG wire#w6
      R_Coil( #Temp )
   END_RUNG
   RUNG wire#w5
      { S7_Templates := "SrcType := Int" } EQ_Contact(in1 := #TemperatureControlSel, in2 := 0)
      I_Contact( #JVDelayTime.TimeOver )
      wire#w7
      S_Coil( #StartJVDelay )
   END_RUNG
   RUNG wire#w7
      R_Coil( #Temp )
   END_RUNG
   // the same network as SCL:
   #_w1 := #Enable AND #Selected AND NOT #RE2;   // rising edge of #Selected
   #RE2 := #Selected;
   IF #_w1 THEN #StartConfirmationPopupTemp := TRUE; END_IF;
   #_w2 := #Enable AND #StartConfirmationPopupTemp AND ((#StartConfirmationPopupSel AND #StartConfirmationAck) OR NOT #StartConfirmationPopupSel);
   IF #_w2 THEN #Started := TRUE; END_IF;
   IF #_w2 AND NOT #JacketPressureSelection AND (#TemperatureControlSel = 1) THEN
       #StartJDDelay := TRUE;
   END_IF;
   IF #_w2 AND NOT #JacketPressureSelection AND (#TemperatureControlSel = 0) THEN
       #StartJVDelay := TRUE;
   END_IF;
   IF #_w2 THEN #StartConfirmationPopupTemp := FALSE; END_IF;
   #_w3 := #Enable AND #Running;
   #StartConfirmationPopup := #_w3 AND #StartConfirmationPopupTemp;
   #EndConfirmationPopup := #_w3 AND #EndConfirmationPopupTemp;
   #JacketAirPurgingPopup := #Enable AND #StartJacketAirPurging AND NOT #EndConfirmationPopupTemp;
   #_w4 := #Enable AND #JacketPressureSelection AND #Temp;
   IF #_w4 AND (#TemperatureControlSel = 1) AND NOT #JDDelayTime.TimeOver THEN
       #StartJDDelay := TRUE;
       #Temp := FALSE;
   END_IF;
   IF #_w4 AND (#TemperatureControlSel = 0) AND NOT #JVDelayTime.TimeOver THEN
       #StartJVDelay := TRUE;
       #Temp := FALSE;
   END_IF;
END_REGION

REGION Network 3: Sensor Selection
   RUNG wire#powerrail
      Contact( #Enable )
      wire#w1
      { S7_Templates := "SrcType := Int" } EQ_Contact(in1 := #SensorSel, in2 := 0)
      Move(in := #ActualTemperatureVessel, out1 => #ActualTemperature)
   END_RUNG
   RUNG wire#w1
      { S7_Templates := "SrcType := Int" } EQ_Contact(in1 := #SensorSel, in2 := 1)
      Move(in := #ActualTemperatureJacket, out1 => #ActualTemperature)
   END_RUNG
   // the same network as SCL:
   IF #Enable AND (#SensorSel = 0) THEN #ActualTemperature := #ActualTemperatureVessel; END_IF;
   IF #Enable AND (#SensorSel = 1) THEN #ActualTemperature := #ActualTemperatureJacket; END_IF;
END_REGION

REGION Network 4: Tolerance
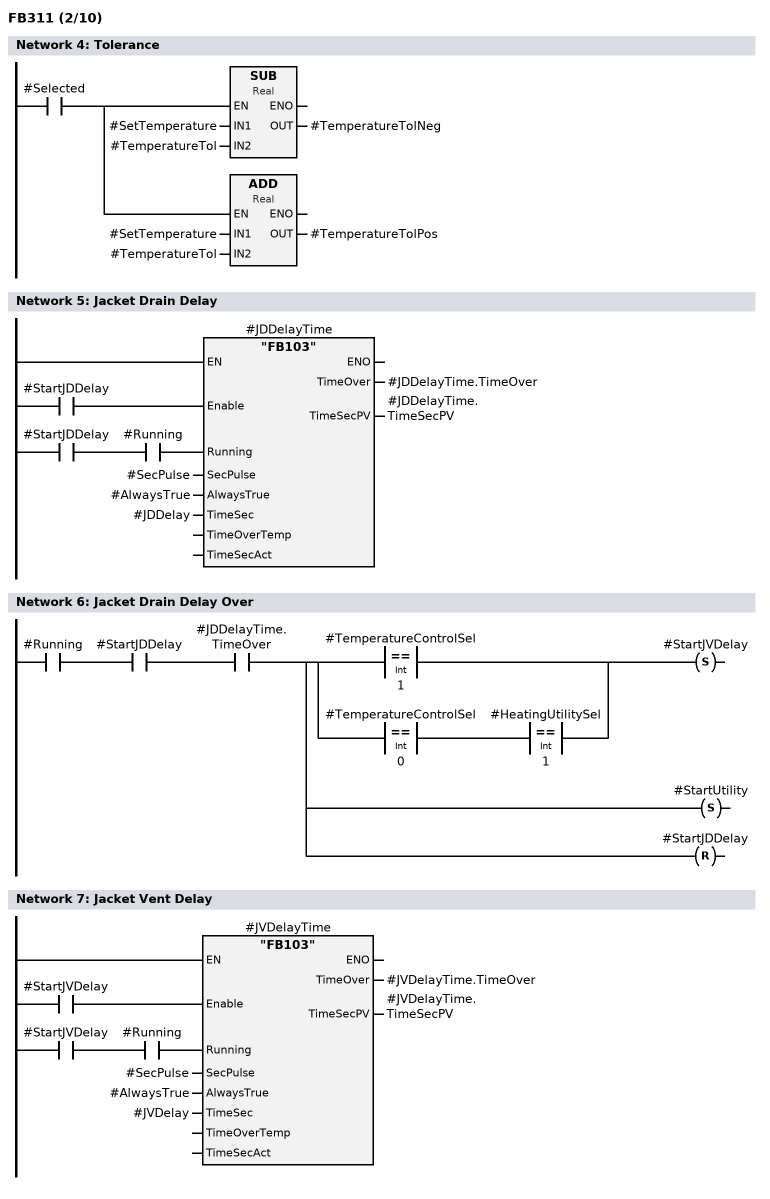
   RUNG wire#powerrail
      Contact( #Selected )
      wire#w1
      { S7_Templates := "SrcType := Real"; S7_GenerateENO := "TRUE" } Sub(in1 := #SetTemperature, in2 := #TemperatureTol, out => #TemperatureTolNeg)
   END_RUNG
   RUNG wire#w1
      { S7_Templates := "SrcType := Real"; S7_GenerateENO := "TRUE" } Add(in1 := #SetTemperature, in2 := #TemperatureTol, out => #TemperatureTolPos)
   END_RUNG
   // the same network as SCL:
   IF #Selected THEN
       #TemperatureTolNeg := #SetTemperature - #TemperatureTol;
       #TemperatureTolPos := #SetTemperature + #TemperatureTol;
   END_IF;
END_REGION

REGION Network 5: Jacket Drain Delay
   RUNG wire#powerrail
      #JDDelayTime(Enable := wire#w1, Running := wire#w2, SecPulse := #SecPulse, AlwaysTrue := #AlwaysTrue, TimeSec := #JDDelay, TimeOverTemp :=, TimeSecAct :=, TimeOver => #JDDelayTime.TimeOver, TimeSecPV => #JDDelayTime.TimeSecPV)
   END_RUNG
   RUNG wire#powerrail
      Contact( #StartJDDelay )
   END_RUNG wire#w1
   RUNG wire#powerrail
      Contact( #StartJDDelay )
      Contact( #Running )
   END_RUNG wire#w2
   // the same network as SCL:
   #JDDelayTime(Enable := #StartJDDelay,   // "FB103"
                Running := #StartJDDelay AND #Running,
                SecPulse := #SecPulse,
                AlwaysTrue := #AlwaysTrue,
                TimeSec := #JDDelay,
                TimeOver => #JDDelayTime.TimeOver,
                TimeSecPV => #JDDelayTime.TimeSecPV);
END_REGION

REGION Network 6: Jacket Drain Delay Over
   RUNG wire#powerrail
      Contact( #Running )
      Contact( #StartJDDelay )
      Contact( #JDDelayTime.TimeOver )
      wire#w1
      { S7_Templates := "SrcType := Int" } EQ_Contact(in1 := #TemperatureControlSel, in2 := 1)
      wire#w2
      S_Coil( #StartJVDelay )
   END_RUNG
   RUNG wire#w1
      { S7_Templates := "SrcType := Int" } EQ_Contact(in1 := #TemperatureControlSel, in2 := 0)
      { S7_Templates := "SrcType := Int" } EQ_Contact(in1 := #HeatingUtilitySel, in2 := 1)
   END_RUNG wire#w2
   RUNG wire#w1
      S_Coil( #StartUtility )
   END_RUNG
   RUNG wire#w1
      R_Coil( #StartJDDelay )
   END_RUNG
   // the same network as SCL:
   #_w1 := #Running AND #StartJDDelay AND #JDDelayTime.TimeOver;
   IF #_w1 AND ((#TemperatureControlSel = 1) OR ((#TemperatureControlSel = 0) AND (#HeatingUtilitySel = 1))) THEN
       #StartJVDelay := TRUE;
   END_IF;
   IF #_w1 THEN
       #StartUtility := TRUE;
       #StartJDDelay := FALSE;
   END_IF;
END_REGION

REGION Network 7: Jacket Vent Delay
   RUNG wire#powerrail
      #JVDelayTime(Enable := wire#w1, Running := wire#w2, SecPulse := #SecPulse, AlwaysTrue := #AlwaysTrue, TimeSec := #JVDelay, TimeOverTemp :=, TimeSecAct :=, TimeOver => #JVDelayTime.TimeOver, TimeSecPV => #JVDelayTime.TimeSecPV)
   END_RUNG
   RUNG wire#powerrail
      Contact( #StartJVDelay )
   END_RUNG wire#w1
   RUNG wire#powerrail
      Contact( #StartJVDelay )
      Contact( #Running )
   END_RUNG wire#w2
   // the same network as SCL:
   #JVDelayTime(Enable := #StartJVDelay,   // "FB103"
                Running := #StartJVDelay AND #Running,
                SecPulse := #SecPulse,
                AlwaysTrue := #AlwaysTrue,
                TimeSec := #JVDelay,
                TimeOver => #JVDelayTime.TimeOver,
                TimeSecPV => #JVDelayTime.TimeSecPV);
END_REGION

REGION Network 8: Jacket Vent Delay Over
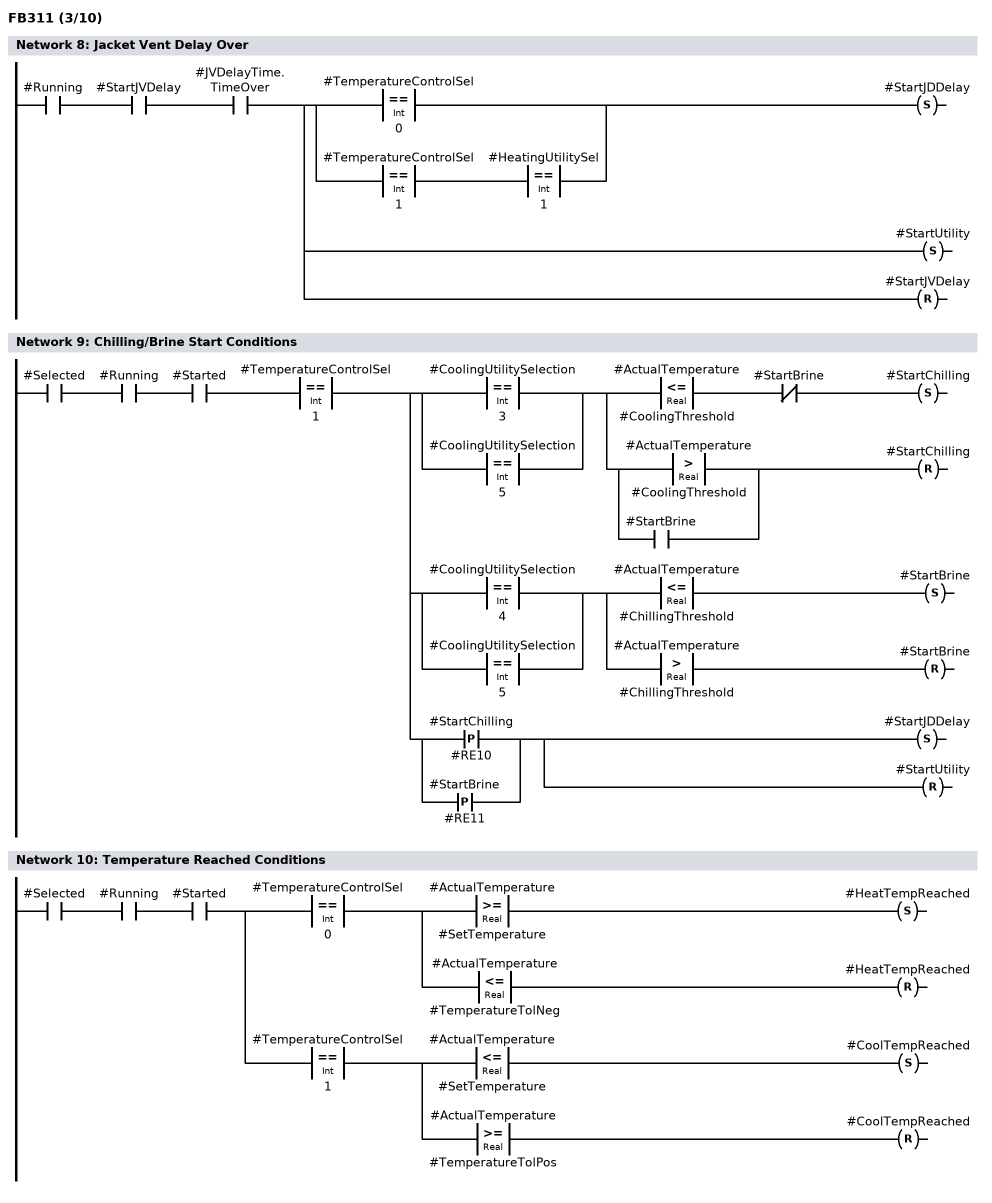
   RUNG wire#powerrail
      Contact( #Running )
      Contact( #StartJVDelay )
      Contact( #JVDelayTime.TimeOver )
      wire#w1
      { S7_Templates := "SrcType := Int" } EQ_Contact(in1 := #TemperatureControlSel, in2 := 0)
      wire#w2
      S_Coil( #StartJDDelay )
   END_RUNG
   RUNG wire#w1
      { S7_Templates := "SrcType := Int" } EQ_Contact(in1 := #TemperatureControlSel, in2 := 1)
      { S7_Templates := "SrcType := Int" } EQ_Contact(in1 := #HeatingUtilitySel, in2 := 1)
   END_RUNG wire#w2
   RUNG wire#w1
      S_Coil( #StartUtility )
   END_RUNG
   RUNG wire#w1
      R_Coil( #StartJVDelay )
   END_RUNG
   // the same network as SCL:
   #_w1 := #Running AND #StartJVDelay AND #JVDelayTime.TimeOver;
   IF #_w1 AND ((#TemperatureControlSel = 0) OR ((#TemperatureControlSel = 1) AND (#HeatingUtilitySel = 1))) THEN
       #StartJDDelay := TRUE;
   END_IF;
   IF #_w1 THEN
       #StartUtility := TRUE;
       #StartJVDelay := FALSE;
   END_IF;
END_REGION

REGION Network 9: Chilling/Brine Start Conditions
   RUNG wire#powerrail
      Contact( #Selected )
      Contact( #Running )
      Contact( #Started )
      { S7_Templates := "SrcType := Int" } EQ_Contact(in1 := #TemperatureControlSel, in2 := 1)
      wire#w1
      { S7_Templates := "SrcType := Int" } EQ_Contact(in1 := #CoolingUtilitySelection, in2 := 3)
      wire#w2
      { S7_Templates := "SrcType := Real" } LE_Contact(in1 := #ActualTemperature, in2 := #CoolingThreshold)
      I_Contact( #StartBrine )
      S_Coil( #StartChilling )
   END_RUNG
   RUNG wire#w1
      { S7_Templates := "SrcType := Int" } EQ_Contact(in1 := #CoolingUtilitySelection, in2 := 5)
   END_RUNG wire#w2
   RUNG wire#w2
      { S7_Templates := "SrcType := Real" } GT_Contact(in1 := #ActualTemperature, in2 := #CoolingThreshold)
      wire#w3
      R_Coil( #StartChilling )
   END_RUNG
   RUNG wire#w2
      Contact( #StartBrine )
   END_RUNG wire#w3
   RUNG wire#w1
      { S7_Templates := "SrcType := Int" } EQ_Contact(in1 := #CoolingUtilitySelection, in2 := 4)
      wire#w4
      { S7_Templates := "SrcType := Real" } LE_Contact(in1 := #ActualTemperature, in2 := #ChillingThreshold)
      S_Coil( #StartBrine )
   END_RUNG
   RUNG wire#w1
      { S7_Templates := "SrcType := Int" } EQ_Contact(in1 := #CoolingUtilitySelection, in2 := 5)
   END_RUNG wire#w4
   RUNG wire#w4
      { S7_Templates := "SrcType := Real" } GT_Contact(in1 := #ActualTemperature, in2 := #ChillingThreshold)
      R_Coil( #StartBrine )
   END_RUNG
   RUNG wire#w1
      P_Contact(operand := #StartChilling, bit := #RE10)
      wire#w5
      S_Coil( #StartJDDelay )
   END_RUNG
   RUNG wire#w1
      P_Contact(operand := #StartBrine, bit := #RE11)
   END_RUNG wire#w5
   RUNG wire#w5
      R_Coil( #StartUtility )
   END_RUNG
   // the same network as SCL:
   #_w1 := #Selected AND #Running AND #Started AND (#TemperatureControlSel = 1);
   #_w2 := #_w1 AND ((#CoolingUtilitySelection = 3) OR (#CoolingUtilitySelection = 5));
   IF #_w2 AND (#ActualTemperature <= #CoolingThreshold) AND NOT #StartBrine THEN
       #StartChilling := TRUE;
   END_IF;
   IF #_w2 AND ((#ActualTemperature > #CoolingThreshold) OR #StartBrine) THEN
       #StartChilling := FALSE;
   END_IF;
   #_w3 := #_w1 AND ((#CoolingUtilitySelection = 4) OR (#CoolingUtilitySelection = 5));
   IF #_w3 AND (#ActualTemperature <= #ChillingThreshold) THEN #StartBrine := TRUE; END_IF;
   IF #_w3 AND (#ActualTemperature > #ChillingThreshold) THEN #StartBrine := FALSE; END_IF;
   #_w4 := #_w1 AND #StartChilling AND NOT #RE10;   // rising edge of #StartChilling
   #RE10 := #StartChilling;
   #_w5 := #_w1 AND #StartBrine AND NOT #RE11;   // rising edge of #StartBrine
   #RE11 := #StartBrine;
   IF #_w4 OR #_w5 THEN
       #StartJDDelay := TRUE;
       #StartUtility := FALSE;
   END_IF;
END_REGION

